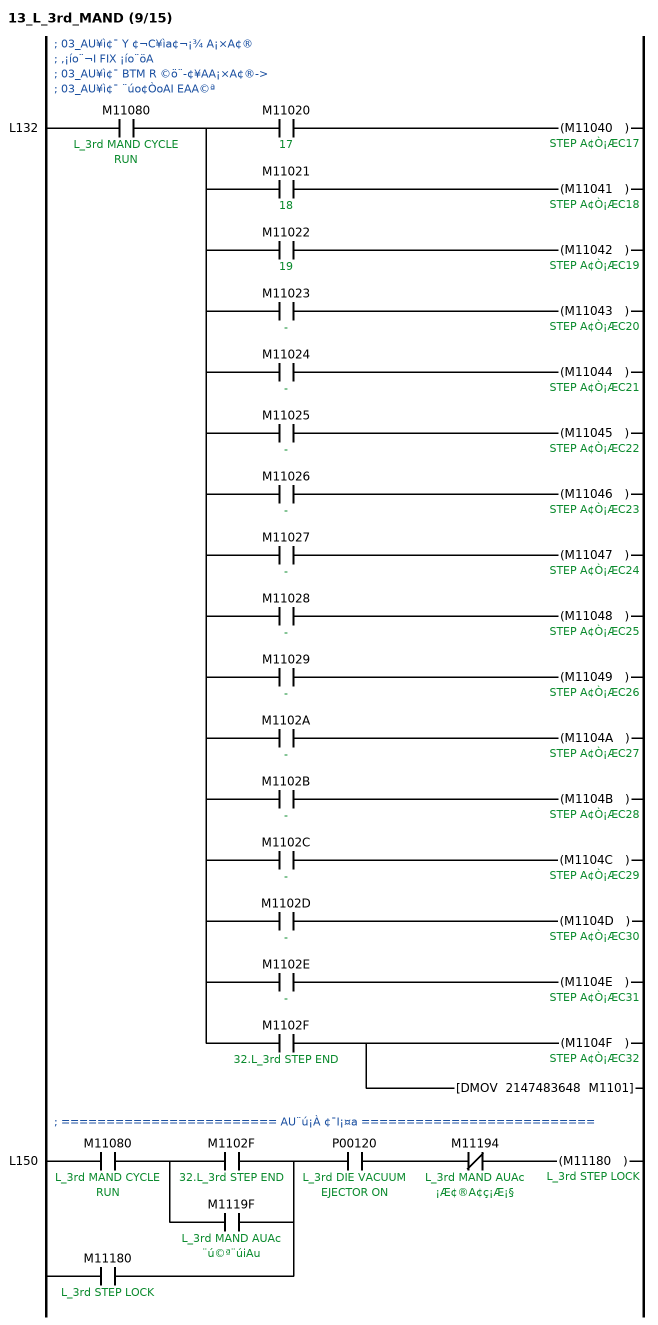
[picture p96: 13_L_3rd_MAND rungs L132-L150]
; L132
LOAD      M11080	// L_3rd MAND CYCLE RUN
MPUSH
AND       M11020	// 17
OUT       M11040	// STEP A¢Ò¡ÆC17
MLOAD
AND       M11021	// 18
OUT       M11041	// STEP A¢Ò¡ÆC18
MLOAD
AND       M11022	// 19
OUT       M11042	// STEP A¢Ò¡ÆC19
MLOAD
AND       M11023	// -
OUT       M11043	// STEP A¢Ò¡ÆC20
MLOAD
AND       M11024	// -
OUT       M11044	// STEP A¢Ò¡ÆC21
MLOAD
AND       M11025	// -
OUT       M11045	// STEP A¢Ò¡ÆC22
MLOAD
AND       M11026	// -
OUT       M11046	// STEP A¢Ò¡ÆC23
MLOAD
AND       M11027	// -
OUT       M11047	// STEP A¢Ò¡ÆC24
MLOAD
AND       M11028	// -
OUT       M11048	// STEP A¢Ò¡ÆC25
MLOAD
AND       M11029	// -
OUT       M11049	// STEP A¢Ò¡ÆC26
MLOAD
AND       M1102A	// -
OUT       M1104A	// STEP A¢Ò¡ÆC27
MLOAD
AND       M1102B	// -
OUT       M1104B	// STEP A¢Ò¡ÆC28
MLOAD
AND       M1102C	// -
OUT       M1104C	// STEP A¢Ò¡ÆC29
MLOAD
AND       M1102D	// -
OUT       M1104D	// STEP A¢Ò¡ÆC30
MLOAD
AND       M1102E	// -
OUT       M1104E	// STEP A¢Ò¡ÆC31
MPOP
AND       M1102F	// 32.L_3rd STEP END
OUT       M1104F	// STEP A¢Ò¡ÆC32
DMOV      2147483648 M1101
// output comment: 03_AU¥ì¢¯ Y ¢¬C¥ìa¢¬¡¾ A¡×A¢® ,¡ío¨¬I FIX ¡ío¨öA
// output comment: 03_AU¥ì¢¯ BTM R ©ö¨­¢¥AA¡×A¢®->
// output comment: 03_AU¥ì¢¯ ¨úo¢ÒoAI EAA©ª
// ======================== AU¨ú¡À ¢¯I¡¤a ==========================
; L150
LOAD      M11080	// L_3rd MAND CYCLE RUN
LOAD      M1102F	// 32.L_3rd STEP END
OR        M1119F	// L_3rd MAND AUAc ¨ú©ª¨úiAu
AND LOAD
OR        M11180	// L_3rd STEP LOCK
AND       P00120	// L_3rd DIE VACUUM EJECTOR ON
AND NOT   M11194	// L_3rd MAND AUAc ¡Æ¢®A¢ç¡Æ¡§
OUT       M11180	// L_3rd STEP LOCK

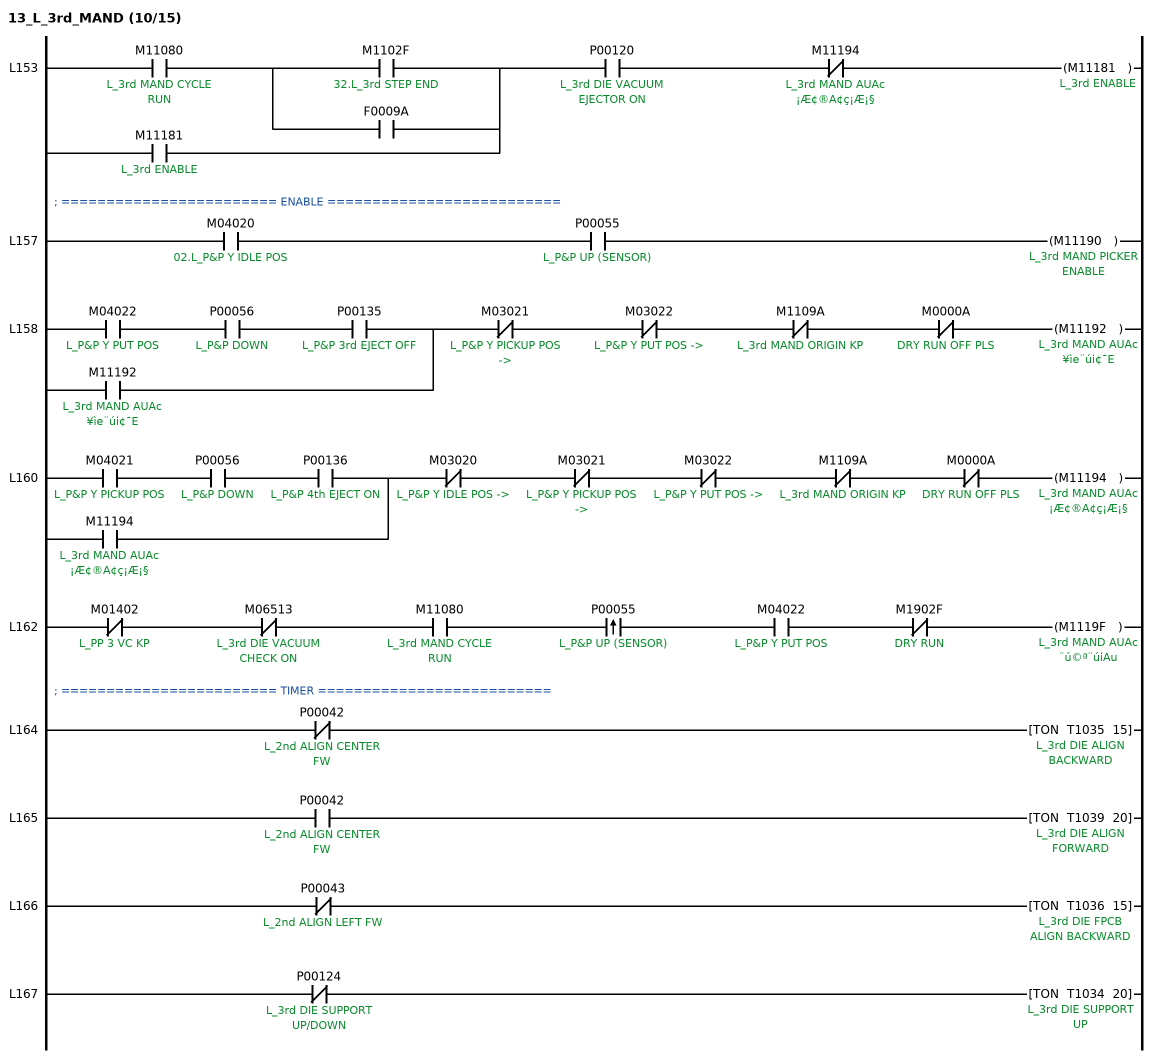
; L153
LOAD      M11080	// L_3rd MAND CYCLE RUN
LOAD      M1102F	// 32.L_3rd STEP END
OR        F0009A
AND LOAD
OR        M11181	// L_3rd ENABLE
AND       P00120	// L_3rd DIE VACUUM EJECTOR ON
AND NOT   M11194	// L_3rd MAND AUAc ¡Æ¢®A¢ç¡Æ¡§
OUT       M11181	// L_3rd ENABLE
// ======================== ENABLE ==========================
; L157
LOAD      M04020	// 02.L_P&P Y IDLE POS
AND       P00055	// L_P&P UP (SENSOR)
OUT       M11190	// L_3rd MAND PICKER ENABLE
; L158
LOAD      M04022	// L_P&P Y PUT POS
AND       P00056	// L_P&P DOWN
AND       P00135	// L_P&P 3rd EJECT OFF
OR        M11192	// L_3rd MAND AUAc ¥ìe¨úi¢¯E
AND NOT   M03021	// L_P&P Y PICKUP POS ->
AND NOT   M03022	// L_P&P Y PUT POS ->
AND NOT   M1109A	// L_3rd MAND ORIGIN KP
AND NOT   M0000A	// DRY RUN OFF PLS
OUT       M11192	// L_3rd MAND AUAc ¥ìe¨úi¢¯E
; L160
LOAD      M04021	// L_P&P Y PICKUP POS
AND       P00056	// L_P&P DOWN
AND       P00136	// L_P&P 4th EJECT ON
OR        M11194	// L_3rd MAND AUAc ¡Æ¢®A¢ç¡Æ¡§
AND NOT   M03020	// L_P&P Y IDLE POS ->
AND NOT   M03021	// L_P&P Y PICKUP POS ->
AND NOT   M03022	// L_P&P Y PUT POS ->
AND NOT   M1109A	// L_3rd MAND ORIGIN KP
AND NOT   M0000A	// DRY RUN OFF PLS
OUT       M11194	// L_3rd MAND AUAc ¡Æ¢®A¢ç¡Æ¡§
; L162
LOAD NOT  M01402	// L_PP 3 VC KP
AND NOT   M06513	// L_3rd DIE VACUUM CHECK ON
AND       M11080	// L_3rd MAND CYCLE RUN
ANDP      P00055	// L_P&P UP (SENSOR)
AND       M04022	// L_P&P Y PUT POS
AND NOT   M1902F	// DRY RUN
OUT       M1119F	// L_3rd MAND AUAc ¨ú©ª¨úiAu
// ======================== TIMER ==========================
; L164
LOAD NOT  P00042	// L_2nd ALIGN CENTER FW
TON       T1035 15	// L_3rd DIE ALIGN BACKWARD
; L165
LOAD      P00042	// L_2nd ALIGN CENTER FW
TON       T1039 20	// L_3rd DIE ALIGN FORWARD
; L166
LOAD NOT  P00043	// L_2nd ALIGN LEFT FW
TON       T1036 15	// L_3rd DIE FPCB ALIGN BACKWARD
; L167
LOAD NOT  P00124	// L_3rd DIE SUPPORT UP/DOWN
TON       T1034 20	// L_3rd DIE SUPPORT UP

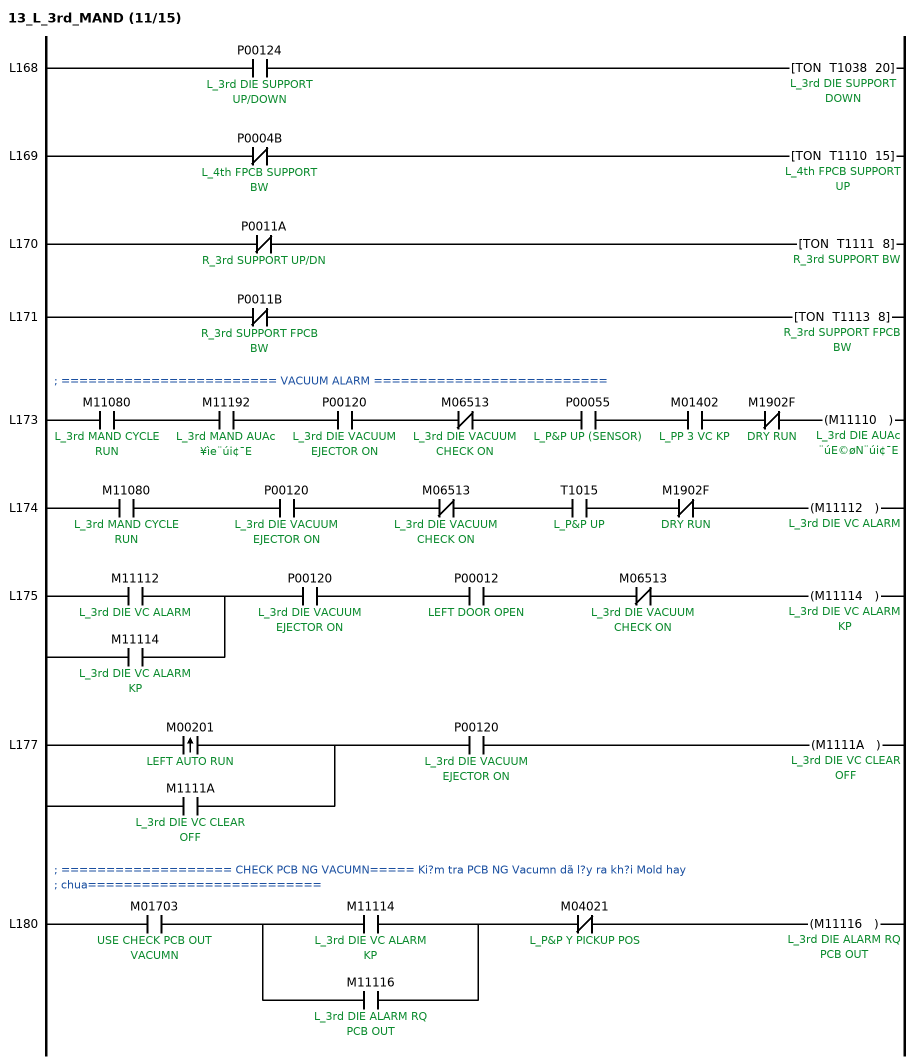
; L168
LOAD      P00124	// L_3rd DIE SUPPORT UP/DOWN
TON       T1038 20	// L_3rd DIE SUPPORT DOWN
; L169
LOAD NOT  P0004B	// L_4th FPCB SUPPORT BW
TON       T1110 15	// L_4th FPCB SUPPORT UP
; L170
LOAD NOT  P0011A	// R_3rd SUPPORT UP/DN
TON       T1111 8	// R_3rd SUPPORT BW
; L171
LOAD NOT  P0011B	// R_3rd SUPPORT FPCB BW
TON       T1113 8	// R_3rd SUPPORT FPCB BW
// ======================== VACUUM ALARM ==========================
; L173
LOAD      M11080	// L_3rd MAND CYCLE RUN
AND       M11192	// L_3rd MAND AUAc ¥ìe¨úi¢¯E
AND       P00120	// L_3rd DIE VACUUM EJECTOR ON
AND NOT   M06513	// L_3rd DIE VACUUM CHECK ON
AND       P00055	// L_P&P UP (SENSOR)
AND       M01402	// L_PP 3 VC KP
AND NOT   M1902F	// DRY RUN
OUT       M11110	// L_3rd DIE AUAc ¨úE©øN¨úi¢¯E
; L174
LOAD      M11080	// L_3rd MAND CYCLE RUN
AND       P00120	// L_3rd DIE VACUUM EJECTOR ON
AND NOT   M06513	// L_3rd DIE VACUUM CHECK ON
AND       T1015	// L_P&P UP
AND NOT   M1902F	// DRY RUN
OUT       M11112	// L_3rd DIE VC ALARM
; L175
LOAD      M11112	// L_3rd DIE VC ALARM
OR        M11114	// L_3rd DIE VC ALARM KP
AND       P00120	// L_3rd DIE VACUUM EJECTOR ON
AND       P00012	// LEFT DOOR OPEN
AND NOT   M06513	// L_3rd DIE VACUUM CHECK ON
OUT       M11114	// L_3rd DIE VC ALARM KP
; L177
LOADP     M00201	// LEFT AUTO RUN
OR        M1111A	// L_3rd DIE VC CLEAR OFF
AND       P00120	// L_3rd DIE VACUUM EJECTOR ON
OUT       M1111A	// L_3rd DIE VC CLEAR OFF
// =================== CHECK PCB NG VACUMN===== Ki?m tra PCB NG Vacumn dã l?y ra kh?i Mold hay chua==========================
; L180
LOAD      M01703	// USE CHECK PCB OUT VACUMN
LOAD      M11114	// L_3rd DIE VC ALARM KP
OR        M11116	// L_3rd DIE ALARM RQ PCB OUT
AND LOAD
AND NOT   M04021	// L_P&P Y PICKUP POS
OUT       M11116	// L_3rd DIE ALARM RQ PCB OUT

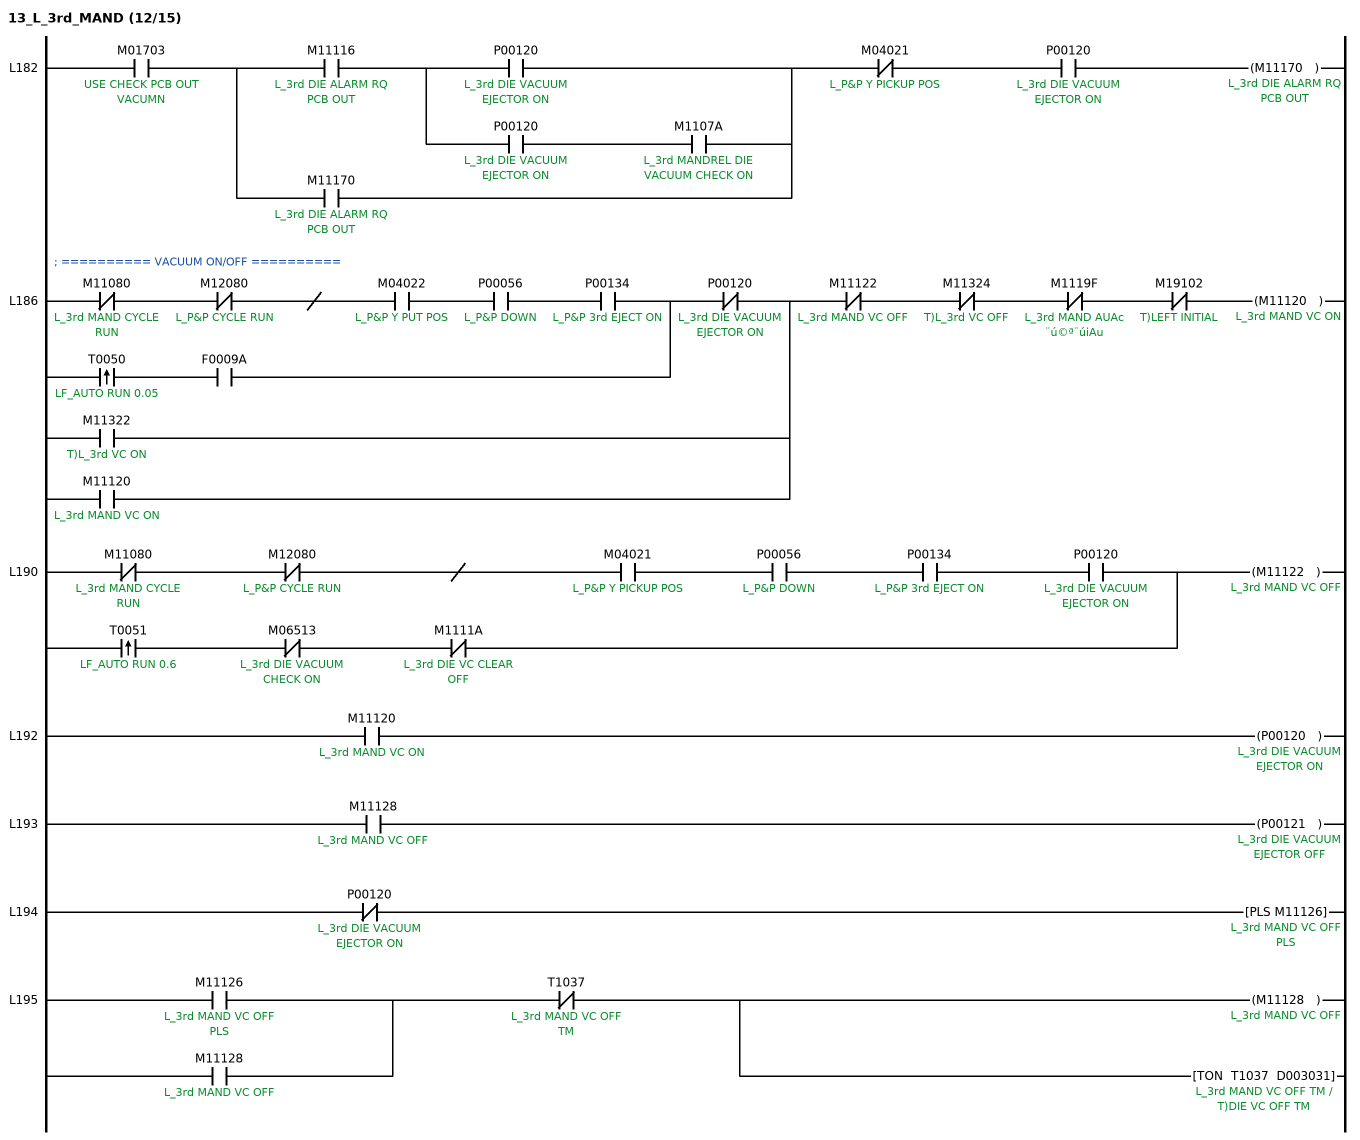
; L182
LOAD      M01703	// USE CHECK PCB OUT VACUMN
LOAD      M11116	// L_3rd DIE ALARM RQ PCB OUT
LOAD      P00120	// L_3rd DIE VACUUM EJECTOR ON
LOAD      P00120	// L_3rd DIE VACUUM EJECTOR ON
AND       M1107A	// L_3rd MANDREL DIE VACUUM CHECK ON
OR LOAD
AND LOAD
OR        M11170	// L_3rd DIE ALARM RQ PCB OUT
AND LOAD
AND NOT   M04021	// L_P&P Y PICKUP POS
AND       P00120	// L_3rd DIE VACUUM EJECTOR ON
OUT       M11170	// L_3rd DIE ALARM RQ PCB OUT
// ========== VACUUM ON/OFF ==========
; L186
LOAD NOT  M11080	// L_3rd MAND CYCLE RUN
AND NOT   M12080	// L_P&P CYCLE RUN
NOT
AND       M04022	// L_P&P Y PUT POS
AND       P00056	// L_P&P DOWN
AND       P00134	// L_P&P 3rd EJECT ON
LOADP     T0050	// LF_AUTO RUN 0.05
AND       F0009A
OR LOAD
AND NOT   P00120	// L_3rd DIE VACUUM EJECTOR ON
OR        M11322	// T)L_3rd VC ON
OR        M11120	// L_3rd MAND VC ON
AND NOT   M11122	// L_3rd MAND VC OFF
AND NOT   M11324	// T)L_3rd VC OFF
AND NOT   M1119F	// L_3rd MAND AUAc ¨ú©ª¨úiAu
AND NOT   M19102	// T)LEFT INITIAL
OUT       M11120	// L_3rd MAND VC ON
; L190
LOAD NOT  M11080	// L_3rd MAND CYCLE RUN
AND NOT   M12080	// L_P&P CYCLE RUN
NOT
AND       M04021	// L_P&P Y PICKUP POS
AND       P00056	// L_P&P DOWN
AND       P00134	// L_P&P 3rd EJECT ON
AND       P00120	// L_3rd DIE VACUUM EJECTOR ON
LOADP     T0051	// LF_AUTO RUN 0.6
AND NOT   M06513	// L_3rd DIE VACUUM CHECK ON
AND NOT   M1111A	// L_3rd DIE VC CLEAR OFF
OR LOAD
OUT       M11122	// L_3rd MAND VC OFF
; L192
LOAD      M11120	// L_3rd MAND VC ON
OUT       P00120	// L_3rd DIE VACUUM EJECTOR ON
; L193
LOAD      M11128	// L_3rd MAND VC OFF
OUT       P00121	// L_3rd DIE VACUUM EJECTOR OFF
; L194
LOAD NOT  P00120	// L_3rd DIE VACUUM EJECTOR ON
OUTP      M11126	// L_3rd MAND VC OFF PLS
; L195
LOAD      M11126	// L_3rd MAND VC OFF PLS
OR        M11128	// L_3rd MAND VC OFF
AND NOT   T1037	// L_3rd MAND VC OFF TM
OUT       M11128	// L_3rd MAND VC OFF
TON       T1037 D003031	// L_3rd MAND VC OFF TM / T)DIE VC OFF TM

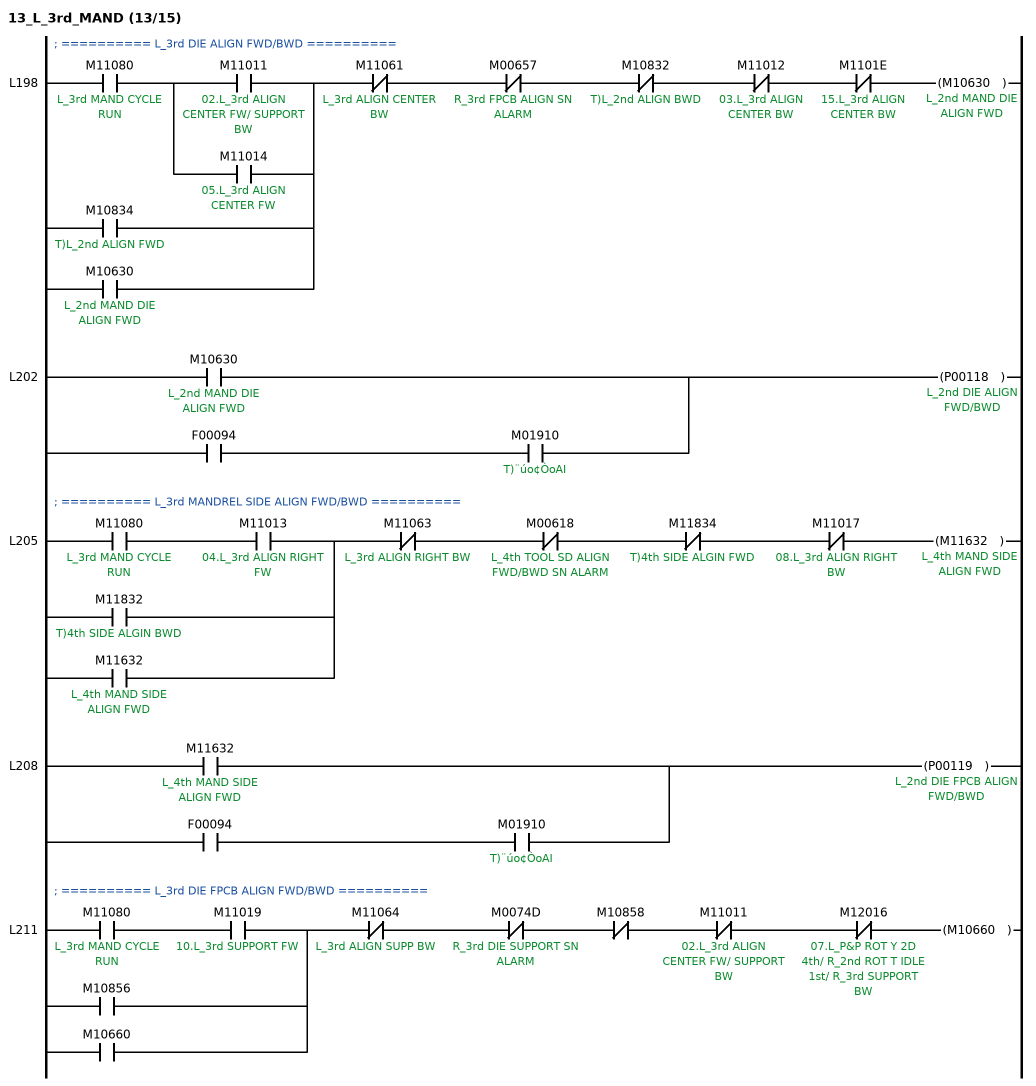
// ========== L_3rd DIE ALIGN FWD/BWD ==========
; L198
LOAD      M11080	// L_3rd MAND CYCLE RUN
LOAD      M11011	// 02.L_3rd ALIGN CENTER FW/ SUPPORT BW
OR        M11014	// 05.L_3rd ALIGN CENTER FW
AND LOAD
OR        M10834	// T)L_2nd ALIGN FWD
OR        M10630	// L_2nd MAND DIE ALIGN FWD
AND NOT   M11061	// L_3rd ALIGN CENTER BW
AND NOT   M00657	// R_3rd FPCB ALIGN SN ALARM
AND NOT   M10832	// T)L_2nd ALIGN BWD
AND NOT   M11012	// 03.L_3rd ALIGN CENTER BW
AND NOT   M1101E	// 15.L_3rd ALIGN CENTER BW
OUT       M10630	// L_2nd MAND DIE ALIGN FWD
; L202
LOAD      M10630	// L_2nd MAND DIE ALIGN FWD
LOAD      F00094
AND       M01910	// T)¨úo¢ÒoAI
OR LOAD
OUT       P00118	// L_2nd DIE ALIGN FWD/BWD
// ========== L_3rd MANDREL SIDE ALIGN FWD/BWD ==========
; L205
LOAD      M11080	// L_3rd MAND CYCLE RUN
AND       M11013	// 04.L_3rd ALIGN RIGHT FW
OR        M11832	// T)4th SIDE ALGIN BWD
OR        M11632	// L_4th MAND SIDE ALIGN FWD
AND NOT   M11063	// L_3rd ALIGN RIGHT BW
AND NOT   M00618	// L_4th TOOL SD ALIGN FWD/BWD SN ALARM
AND NOT   M11834	// T)4th SIDE ALGIN FWD
AND NOT   M11017	// 08.L_3rd ALIGN RIGHT BW
OUT       M11632	// L_4th MAND SIDE ALIGN FWD
; L208
LOAD      M11632	// L_4th MAND SIDE ALIGN FWD
LOAD      F00094
AND       M01910	// T)¨úo¢ÒoAI
OR LOAD
OUT       P00119	// L_2nd DIE FPCB ALIGN FWD/BWD
// ========== L_3rd DIE FPCB ALIGN FWD/BWD ==========
; L211
LOAD      M11080	// L_3rd MAND CYCLE RUN
AND       M11019	// 10.L_3rd SUPPORT FW
OR        M10856
OR        M10660
AND NOT   M11064	// L_3rd ALIGN SUPP BW
AND NOT   M0074D	// R_3rd DIE SUPPORT SN ALARM
AND NOT   M10858
AND NOT   M11011	// 02.L_3rd ALIGN CENTER FW/ SUPPORT BW
AND NOT   M12016	// 07.L_P&P ROT Y 2D 4th/ R_2nd ROT T IDLE 1st/ R_3rd SUPPORT BW
OUT       M10660

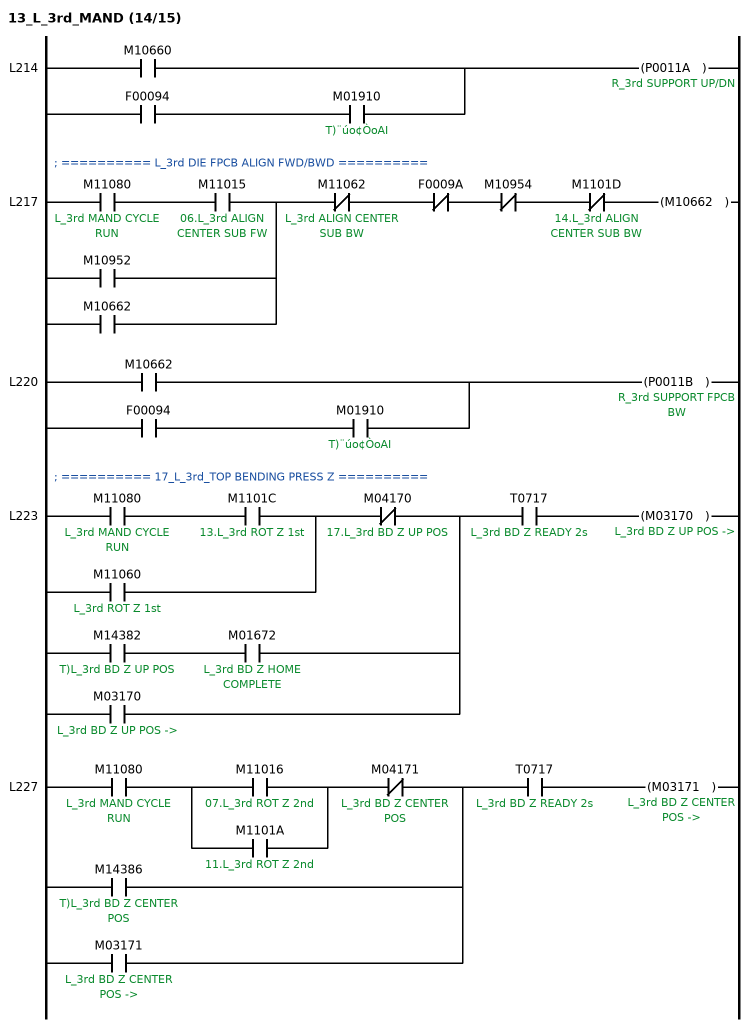
; L214
LOAD      M10660
LOAD      F00094
AND       M01910	// T)¨úo¢ÒoAI
OR LOAD
OUT       P0011A	// R_3rd SUPPORT UP/DN
// ========== L_3rd DIE FPCB ALIGN FWD/BWD ==========
; L217
LOAD      M11080	// L_3rd MAND CYCLE RUN
AND       M11015	// 06.L_3rd ALIGN CENTER SUB FW
OR        M10952
OR        M10662
AND NOT   M11062	// L_3rd ALIGN CENTER SUB BW
AND NOT   F0009A
AND NOT   M10954
AND NOT   M1101D	// 14.L_3rd ALIGN CENTER SUB BW
OUT       M10662
; L220
LOAD      M10662
LOAD      F00094
AND       M01910	// T)¨úo¢ÒoAI
OR LOAD
OUT       P0011B	// R_3rd SUPPORT FPCB BW
// ========== 17_L_3rd_TOP BENDING PRESS Z ==========
; L223
LOAD      M11080	// L_3rd MAND CYCLE RUN
AND       M1101C	// 13.L_3rd ROT Z 1st
OR        M11060	// L_3rd ROT Z 1st
AND NOT   M04170	// 17.L_3rd BD Z UP POS
LOAD      M14382	// T)L_3rd BD Z UP POS
AND       M01672	// L_3rd BD Z HOME COMPLETE
OR LOAD
OR        M03170	// L_3rd BD Z UP POS ->
AND       T0717	// L_3rd BD Z READY 2s
OUT       M03170	// L_3rd BD Z UP POS ->
; L227
LOAD      M11080	// L_3rd MAND CYCLE RUN
LOAD      M11016	// 07.L_3rd ROT Z 2nd
OR        M1101A	// 11.L_3rd ROT Z 2nd
AND LOAD
AND NOT   M04171	// L_3rd BD Z CENTER POS
OR        M14386	// T)L_3rd BD Z CENTER POS
OR        M03171	// L_3rd BD Z CENTER POS ->
AND       T0717	// L_3rd BD Z READY 2s
OUT       M03171	// L_3rd BD Z CENTER POS ->

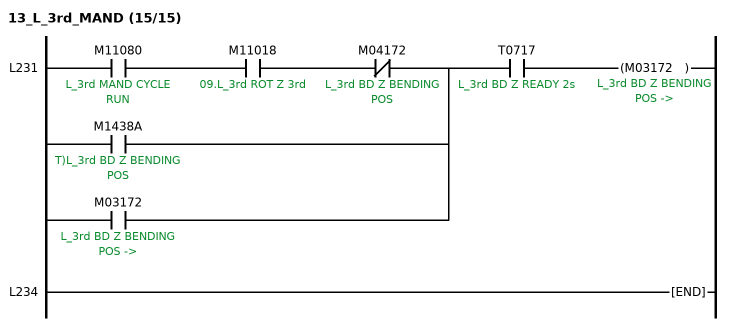
; L231
LOAD      M11080	// L_3rd MAND CYCLE RUN
AND       M11018	// 09.L_3rd ROT Z 3rd
AND NOT   M04172	// L_3rd BD Z BENDING POS
OR        M1438A	// T)L_3rd BD Z BENDING POS
OR        M03172	// L_3rd BD Z BENDING POS ->
AND       T0717	// L_3rd BD Z READY 2s
OUT       M03172	// L_3rd BD Z BENDING POS ->
; L234
END

PROGRAM 14_L_TOOL (task: ¨ö¨¬A¥ì CA¡¤I¡¾¡¿¡¤¡Í)

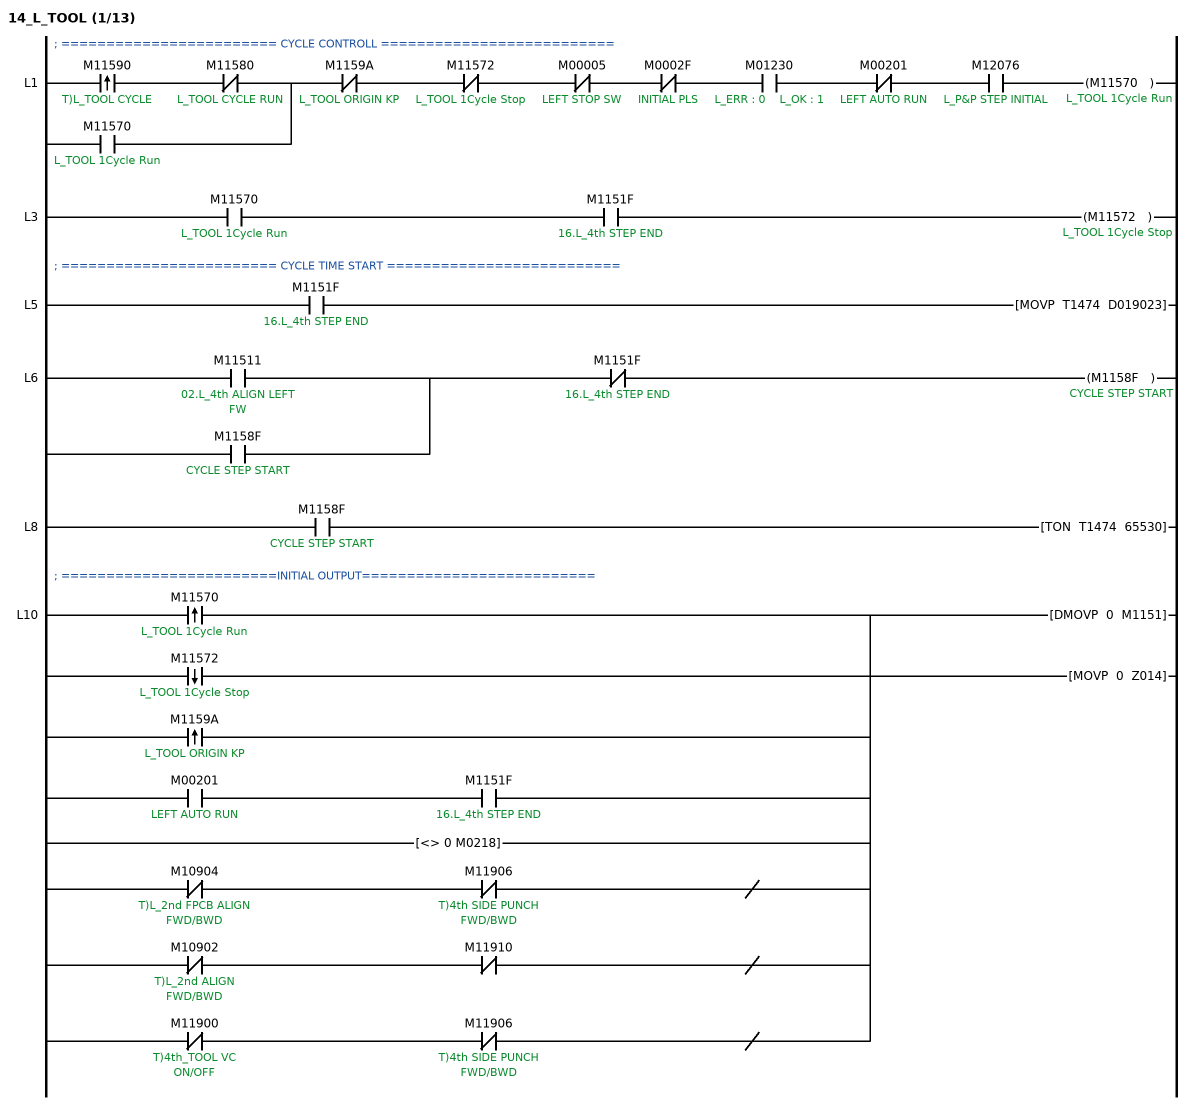
// ======================== CYCLE CONTROLL ==========================
; L1
LOADP     M11590	// T)L_TOOL CYCLE
AND NOT   M11580	// L_TOOL CYCLE RUN
OR        M11570	// L_TOOL 1Cycle Run
AND NOT   M1159A	// L_TOOL ORIGIN KP
AND NOT   M11572	// L_TOOL 1Cycle Stop
AND NOT   M00005	// LEFT STOP SW
AND NOT   M0002F	// INITIAL PLS
AND       M01230	// L_ERR : 0    L_OK : 1
AND NOT   M00201	// LEFT AUTO RUN
AND       M12076	// L_P&P STEP INITIAL
OUT       M11570	// L_TOOL 1Cycle Run
; L3
LOAD      M11570	// L_TOOL 1Cycle Run
AND       M1151F	// 16.L_4th STEP END
OUT       M11572	// L_TOOL 1Cycle Stop
// ======================== CYCLE TIME START ==========================
; L5
LOAD      M1151F	// 16.L_4th STEP END
MOVP      T1474 D019023
; L6
LOAD      M11511	// 02.L_4th ALIGN LEFT FW
OR        M1158F	// CYCLE STEP START
AND NOT   M1151F	// 16.L_4th STEP END
OUT       M1158F	// CYCLE STEP START
; L8
LOAD      M1158F	// CYCLE STEP START
TON       T1474 65530
// ========================INITIAL OUTPUT==========================
; L10
LOADP     M11570	// L_TOOL 1Cycle Run
ORN       M11572	// L_TOOL 1Cycle Stop
ORP       M1159A	// L_TOOL ORIGIN KP
LOAD      M00201	// LEFT AUTO RUN
AND       M1151F	// 16.L_4th STEP END
OR LOAD
OR<>      0 M0218
LOAD NOT  M10904	// T)L_2nd FPCB ALIGN FWD/BWD
AND NOT   M11906	// T)4th SIDE PUNCH FWD/BWD
NOT
OR LOAD
LOAD NOT  M10902	// T)L_2nd ALIGN FWD/BWD
AND NOT   M11910
NOT
OR LOAD
LOAD NOT  M11900	// T)4th_TOOL VC ON/OFF
AND NOT   M11906	// T)4th SIDE PUNCH FWD/BWD
NOT
OR LOAD
DMOVP     0 M1151
MOVP      0 Z014

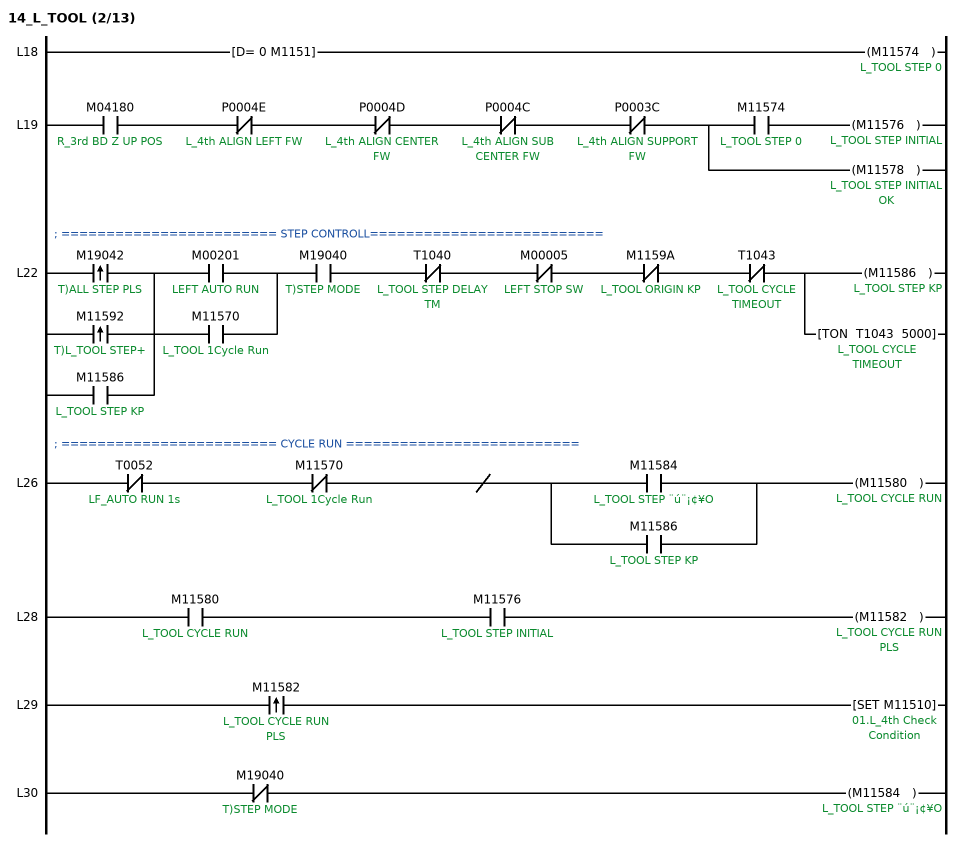
; L18
LOADD=    0 M1151
OUT       M11574	// L_TOOL STEP 0
; L19
LOAD      M04180	// R_3rd BD Z UP POS
AND NOT   P0004E	// L_4th ALIGN LEFT FW
AND NOT   P0004D	// L_4th ALIGN CENTER FW
AND NOT   P0004C	// L_4th ALIGN SUB CENTER FW
AND NOT   P0003C	// L_4th ALIGN SUPPORT FW
MPUSH
AND       M11574	// L_TOOL STEP 0
OUT       M11576	// L_TOOL STEP INITIAL
MPOP
OUT       M11578	// L_TOOL STEP INITIAL OK
// ======================== STEP CONTROLL==========================
; L22
LOADP     M19042	// T)ALL STEP PLS
ORP       M11592	// T)L_TOOL STEP+
OR        M11586	// L_TOOL STEP KP
LOAD      M00201	// LEFT AUTO RUN
OR        M11570	// L_TOOL 1Cycle Run
AND LOAD
AND       M19040	// T)STEP MODE
AND NOT   T1040	// L_TOOL STEP DELAY TM
AND NOT   M00005	// LEFT STOP SW
AND NOT   M1159A	// L_TOOL ORIGIN KP
AND NOT   T1043	// L_TOOL CYCLE TIMEOUT
OUT       M11586	// L_TOOL STEP KP
TON       T1043 5000	// L_TOOL CYCLE TIMEOUT
// ======================== CYCLE RUN ==========================
; L26
LOAD NOT  T0052	// LF_AUTO RUN 1s
AND NOT   M11570	// L_TOOL 1Cycle Run
NOT
LOAD      M11584	// L_TOOL STEP ¨ú¨¡¢¥O
OR        M11586	// L_TOOL STEP KP
AND LOAD
OUT       M11580	// L_TOOL CYCLE RUN
; L28
LOAD      M11580	// L_TOOL CYCLE RUN
AND       M11576	// L_TOOL STEP INITIAL
OUT       M11582	// L_TOOL CYCLE RUN PLS
; L29
LOADP     M11582	// L_TOOL CYCLE RUN PLS
SET       M11510	// 01.L_4th Check Condition
; L30
LOAD NOT  M19040	// T)STEP MODE
OUT       M11584	// L_TOOL STEP ¨ú¨¡¢¥O

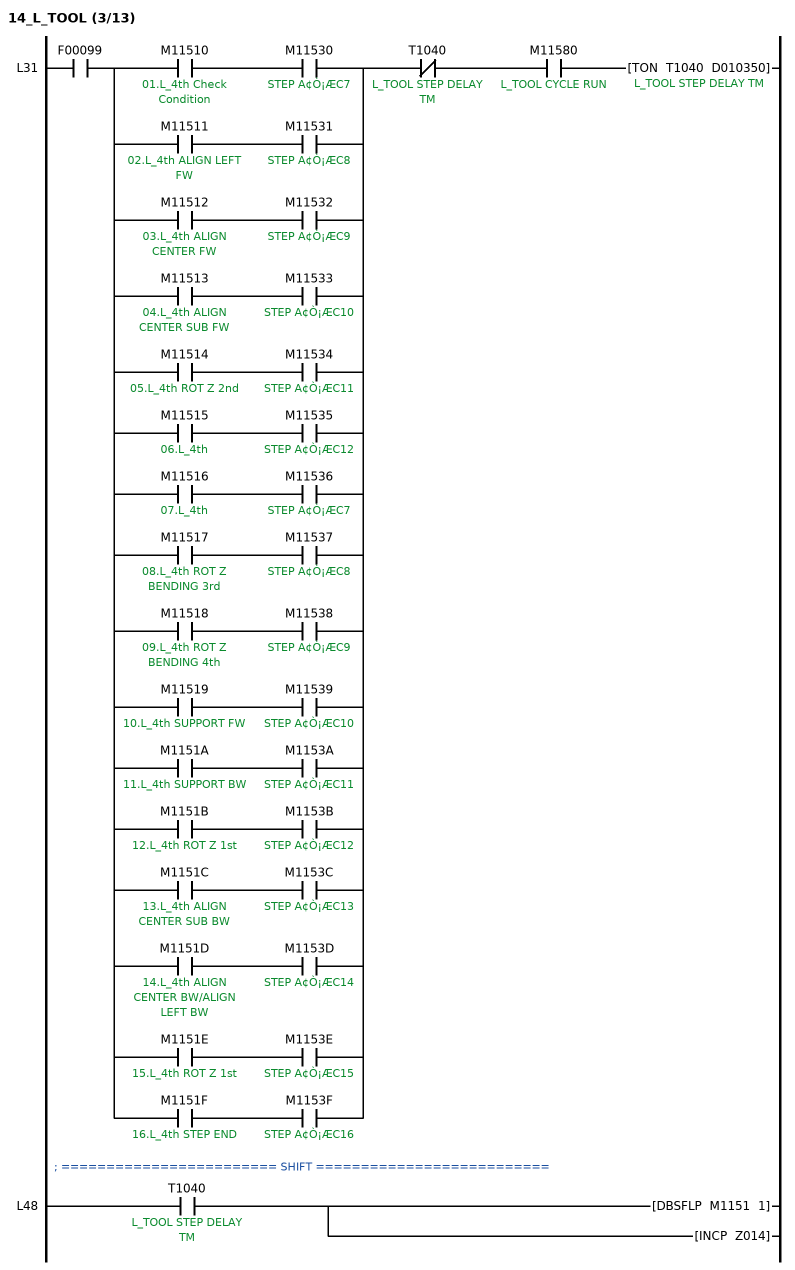
; L31
LOAD      F00099
LOAD      M11510	// 01.L_4th Check Condition
AND       M11530	// STEP A¢Ò¡ÆC7
LOAD      M11511	// 02.L_4th ALIGN LEFT FW
AND       M11531	// STEP A¢Ò¡ÆC8
OR LOAD
LOAD      M11512	// 03.L_4th ALIGN CENTER FW
AND       M11532	// STEP A¢Ò¡ÆC9
OR LOAD
LOAD      M11513	// 04.L_4th ALIGN CENTER SUB FW
AND       M11533	// STEP A¢Ò¡ÆC10
OR LOAD
LOAD      M11514	// 05.L_4th ROT Z 2nd
AND       M11534	// STEP A¢Ò¡ÆC11
OR LOAD
LOAD      M11515	// 06.L_4th 
AND       M11535	// STEP A¢Ò¡ÆC12
OR LOAD
LOAD      M11516	// 07.L_4th 
AND       M11536	// STEP A¢Ò¡ÆC7
OR LOAD
LOAD      M11517	// 08.L_4th ROT Z BENDING 3rd
AND       M11537	// STEP A¢Ò¡ÆC8
OR LOAD
LOAD      M11518	// 09.L_4th ROT Z BENDING 4th
AND       M11538	// STEP A¢Ò¡ÆC9
OR LOAD
LOAD      M11519	// 10.L_4th SUPPORT FW
AND       M11539	// STEP A¢Ò¡ÆC10
OR LOAD
LOAD      M1151A	// 11.L_4th SUPPORT BW
AND       M1153A	// STEP A¢Ò¡ÆC11
OR LOAD
LOAD      M1151B	// 12.L_4th ROT Z 1st
AND       M1153B	// STEP A¢Ò¡ÆC12
OR LOAD
LOAD      M1151C	// 13.L_4th ALIGN CENTER SUB BW
AND       M1153C	// STEP A¢Ò¡ÆC13
OR LOAD
LOAD      M1151D	// 14.L_4th ALIGN CENTER BW/ALIGN LEFT BW
AND       M1153D	// STEP A¢Ò¡ÆC14
OR LOAD
LOAD      M1151E	// 15.L_4th ROT Z 1st
AND       M1153E	// STEP A¢Ò¡ÆC15
OR LOAD
LOAD      M1151F	// 16.L_4th STEP END
AND       M1153F	// STEP A¢Ò¡ÆC16
OR LOAD
AND LOAD
AND NOT   T1040	// L_TOOL STEP DELAY TM
AND       M11580	// L_TOOL CYCLE RUN
TON       T1040 D010350	// L_TOOL STEP DELAY TM
// ======================== SHIFT ==========================
; L48
LOAD      T1040	// L_TOOL STEP DELAY TM
DBSFLP    M1151 1
INCP      Z014

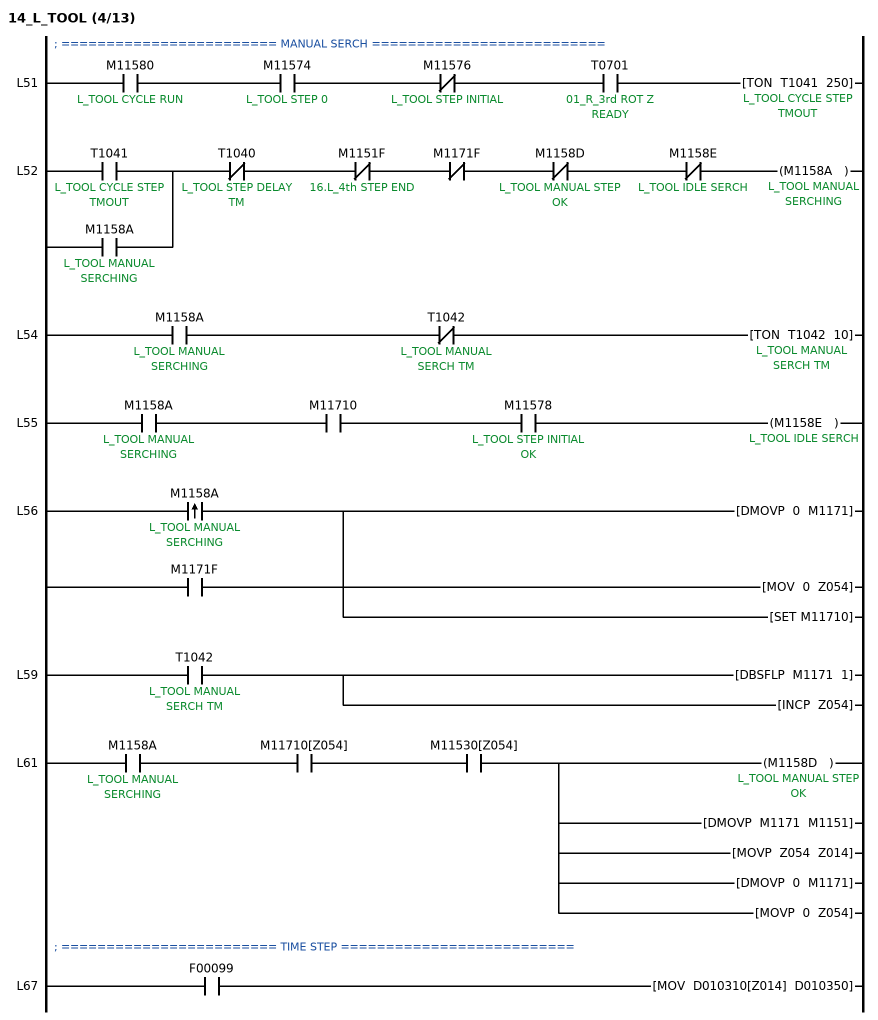
// ======================== MANUAL SERCH ==========================
; L51
LOAD      M11580	// L_TOOL CYCLE RUN
AND       M11574	// L_TOOL STEP 0
AND NOT   M11576	// L_TOOL STEP INITIAL
AND       T0701	// 01_R_3rd ROT Z READY
TON       T1041 250	// L_TOOL CYCLE STEP TMOUT
; L52
LOAD      T1041	// L_TOOL CYCLE STEP TMOUT
OR        M1158A	// L_TOOL MANUAL SERCHING
AND NOT   T1040	// L_TOOL STEP DELAY TM
AND NOT   M1151F	// 16.L_4th STEP END
AND NOT   M1171F
AND NOT   M1158D	// L_TOOL MANUAL STEP OK
AND NOT   M1158E	// L_TOOL IDLE SERCH
OUT       M1158A	// L_TOOL MANUAL SERCHING
; L54
LOAD      M1158A	// L_TOOL MANUAL SERCHING
AND NOT   T1042	// L_TOOL MANUAL SERCH TM
TON       T1042 10	// L_TOOL MANUAL SERCH TM
; L55
LOAD      M1158A	// L_TOOL MANUAL SERCHING
AND       M11710
AND       M11578	// L_TOOL STEP INITIAL OK
OUT       M1158E	// L_TOOL IDLE SERCH
; L56
LOADP     M1158A	// L_TOOL MANUAL SERCHING
OR        M1171F
DMOVP     0 M1171
MOV       0 Z054
SET       M11710
; L59
LOAD      T1042	// L_TOOL MANUAL SERCH TM
DBSFLP    M1171 1
INCP      Z054
; L61
LOAD      M1158A	// L_TOOL MANUAL SERCHING
AND       M11710[Z054]
AND       M11530[Z054]
OUT       M1158D	// L_TOOL MANUAL STEP OK
DMOVP     M1171 M1151
MOVP      Z054 Z014
DMOVP     0 M1171
MOVP      0 Z054
// ======================== TIME STEP ==========================
; L67
LOAD      F00099
MOV       D010310[Z014] D010350

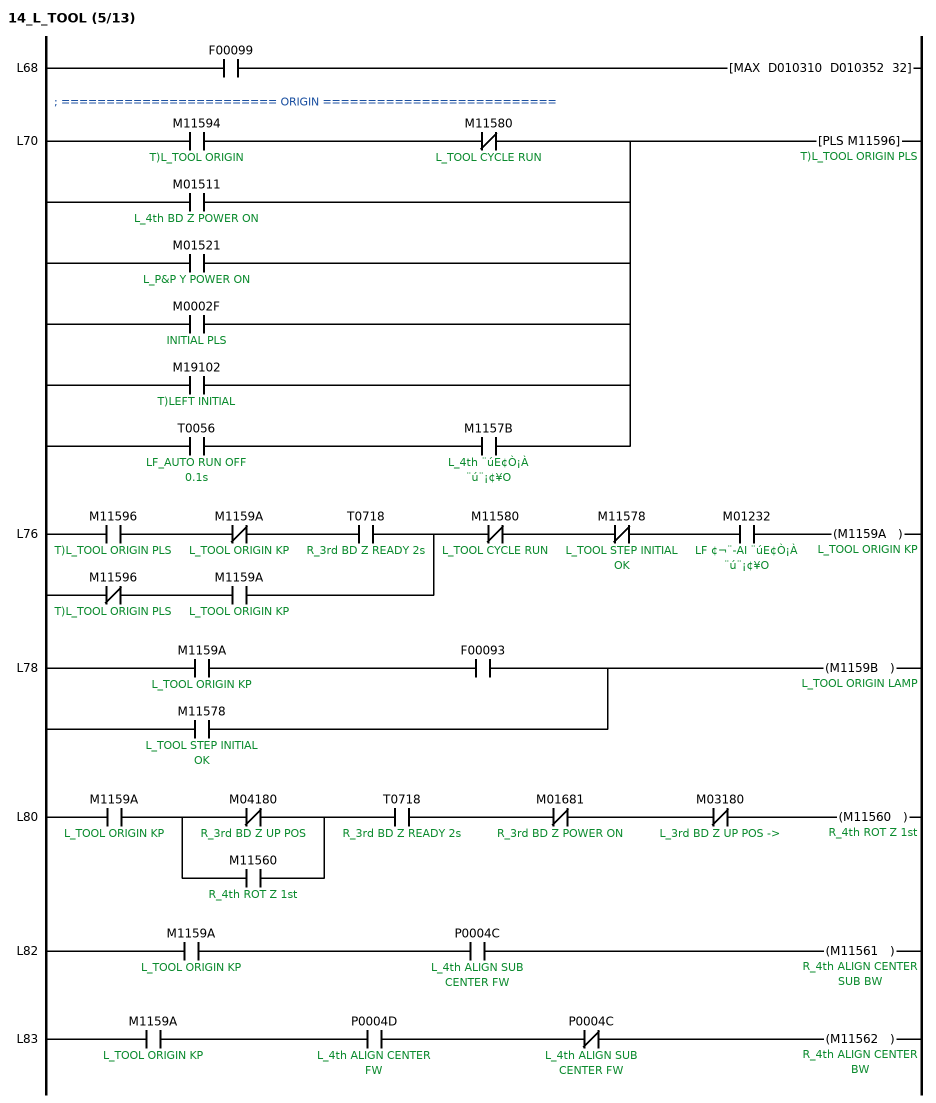
; L68
LOAD      F00099
MAX       D010310 D010352 32
// ======================== ORIGIN ==========================
; L70
LOAD      M11594	// T)L_TOOL ORIGIN
AND NOT   M11580	// L_TOOL CYCLE RUN
OR        M01511	// L_4th BD Z POWER ON
OR        M01521	// L_P&P Y POWER ON
OR        M0002F	// INITIAL PLS
OR        M19102	// T)LEFT INITIAL
LOAD      T0056	// LF_AUTO RUN OFF 0.1s
AND       M1157B	// L_4th ¨úE¢Ò¡À ¨ú¨¡¢¥O
OR LOAD
OUTP      M11596	// T)L_TOOL ORIGIN PLS
; L76
LOAD      M11596	// T)L_TOOL ORIGIN PLS
AND NOT   M1159A	// L_TOOL ORIGIN KP
AND       T0718	// R_3rd BD Z READY 2s
LOAD NOT  M11596	// T)L_TOOL ORIGIN PLS
AND       M1159A	// L_TOOL ORIGIN KP
OR LOAD
AND NOT   M11580	// L_TOOL CYCLE RUN
AND NOT   M11578	// L_TOOL STEP INITIAL OK
AND       M01232	// LF ¢¬¨­AI ¨úE¢Ò¡À ¨ú¨¡¢¥O
OUT       M1159A	// L_TOOL ORIGIN KP
; L78
LOAD      M1159A	// L_TOOL ORIGIN KP
AND       F00093
OR        M11578	// L_TOOL STEP INITIAL OK
OUT       M1159B	// L_TOOL ORIGIN LAMP
; L80
LOAD      M1159A	// L_TOOL ORIGIN KP
LOAD NOT  M04180	// R_3rd BD Z UP POS
OR        M11560	// R_4th ROT Z 1st
AND LOAD
AND       T0718	// R_3rd BD Z READY 2s
AND NOT   M01681	// R_3rd BD Z POWER ON
AND NOT   M03180	// L_3rd BD Z UP POS ->
OUT       M11560	// R_4th ROT Z 1st
; L82
LOAD      M1159A	// L_TOOL ORIGIN KP
AND       P0004C	// L_4th ALIGN SUB CENTER FW
OUT       M11561	// R_4th ALIGN CENTER SUB BW
; L83
LOAD      M1159A	// L_TOOL ORIGIN KP
AND       P0004D	// L_4th ALIGN CENTER FW
AND NOT   P0004C	// L_4th ALIGN SUB CENTER FW
OUT       M11562	// R_4th ALIGN CENTER BW

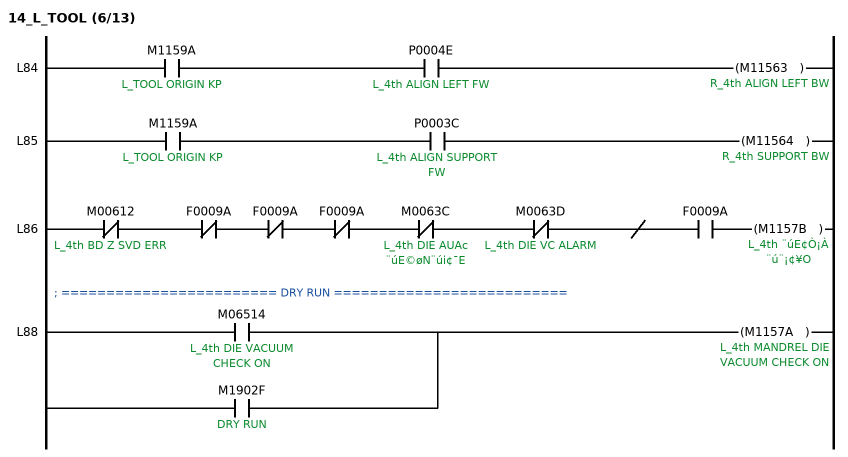
; L84
LOAD      M1159A	// L_TOOL ORIGIN KP
AND       P0004E	// L_4th ALIGN LEFT FW
OUT       M11563	// R_4th ALIGN LEFT BW
; L85
LOAD      M1159A	// L_TOOL ORIGIN KP
AND       P0003C	// L_4th ALIGN SUPPORT FW
OUT       M11564	// R_4th SUPPORT BW
; L86
LOAD NOT  M00612	// L_4th BD Z SVD ERR
AND NOT   F0009A
AND NOT   F0009A
AND NOT   F0009A
AND NOT   M0063C	// L_4th DIE AUAc ¨úE©øN¨úi¢¯E
AND NOT   M0063D	// L_4th DIE VC ALARM
NOT
AND       F0009A
OUT       M1157B	// L_4th ¨úE¢Ò¡À ¨ú¨¡¢¥O
// ======================== DRY RUN ==========================
; L88
LOAD      M06514	// L_4th DIE VACUUM CHECK ON
OR        M1902F	// DRY RUN
OUT       M1157A	// L_4th MANDREL DIE VACUUM CHECK ON

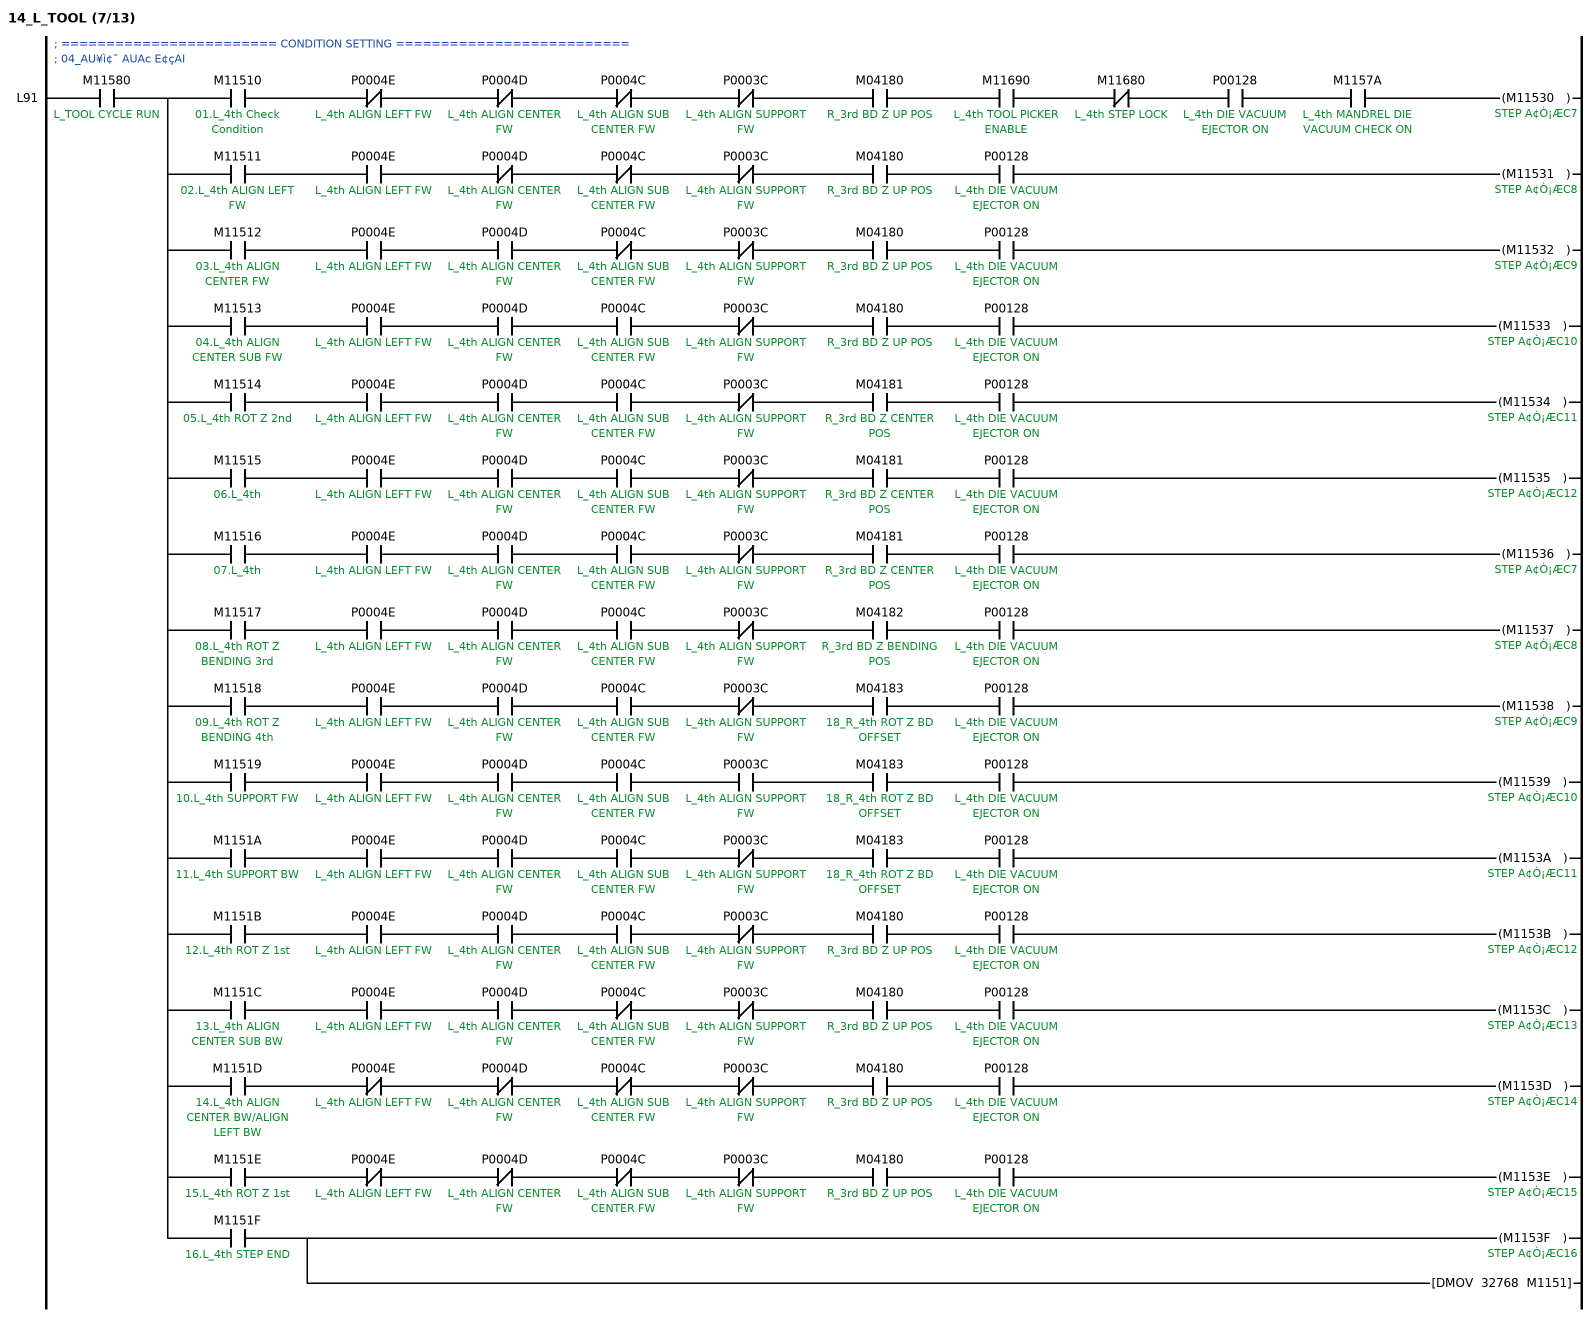
// ======================== CONDITION SETTING ==========================
; L91
LOAD      M11580	// L_TOOL CYCLE RUN
MPUSH
AND       M11510	// 01.L_4th Check Condition
AND NOT   P0004E	// L_4th ALIGN LEFT FW
AND NOT   P0004D	// L_4th ALIGN CENTER FW
AND NOT   P0004C	// L_4th ALIGN SUB CENTER FW
AND NOT   P0003C	// L_4th ALIGN SUPPORT FW
AND       M04180	// R_3rd BD Z UP POS
AND       M11690	// L_4th TOOL PICKER ENABLE
AND NOT   M11680	// L_4th STEP LOCK
AND       P00128	// L_4th DIE VACUUM EJECTOR ON
AND       M1157A	// L_4th MANDREL DIE VACUUM CHECK ON
OUT       M11530	// STEP A¢Ò¡ÆC7
MLOAD
AND       M11511	// 02.L_4th ALIGN LEFT FW
AND       P0004E	// L_4th ALIGN LEFT FW
AND NOT   P0004D	// L_4th ALIGN CENTER FW
AND NOT   P0004C	// L_4th ALIGN SUB CENTER FW
AND NOT   P0003C	// L_4th ALIGN SUPPORT FW
AND       M04180	// R_3rd BD Z UP POS
AND       P00128	// L_4th DIE VACUUM EJECTOR ON
OUT       M11531	// STEP A¢Ò¡ÆC8
MLOAD
AND       M11512	// 03.L_4th ALIGN CENTER FW
AND       P0004E	// L_4th ALIGN LEFT FW
AND       P0004D	// L_4th ALIGN CENTER FW
AND NOT   P0004C	// L_4th ALIGN SUB CENTER FW
AND NOT   P0003C	// L_4th ALIGN SUPPORT FW
AND       M04180	// R_3rd BD Z UP POS
AND       P00128	// L_4th DIE VACUUM EJECTOR ON
OUT       M11532	// STEP A¢Ò¡ÆC9
MLOAD
AND       M11513	// 04.L_4th ALIGN CENTER SUB FW
AND       P0004E	// L_4th ALIGN LEFT FW
AND       P0004D	// L_4th ALIGN CENTER FW
AND       P0004C	// L_4th ALIGN SUB CENTER FW
AND NOT   P0003C	// L_4th ALIGN SUPPORT FW
AND       M04180	// R_3rd BD Z UP POS
AND       P00128	// L_4th DIE VACUUM EJECTOR ON
OUT       M11533	// STEP A¢Ò¡ÆC10
MLOAD
AND       M11514	// 05.L_4th ROT Z 2nd
AND       P0004E	// L_4th ALIGN LEFT FW
AND       P0004D	// L_4th ALIGN CENTER FW
AND       P0004C	// L_4th ALIGN SUB CENTER FW
AND NOT   P0003C	// L_4th ALIGN SUPPORT FW
AND       M04181	// R_3rd BD Z CENTER POS
AND       P00128	// L_4th DIE VACUUM EJECTOR ON
OUT       M11534	// STEP A¢Ò¡ÆC11
MLOAD
AND       M11515	// 06.L_4th 
AND       P0004E	// L_4th ALIGN LEFT FW
AND       P0004D	// L_4th ALIGN CENTER FW
AND       P0004C	// L_4th ALIGN SUB CENTER FW
AND NOT   P0003C	// L_4th ALIGN SUPPORT FW
AND       M04181	// R_3rd BD Z CENTER POS
AND       P00128	// L_4th DIE VACUUM EJECTOR ON
OUT       M11535	// STEP A¢Ò¡ÆC12
MLOAD
AND       M11516	// 07.L_4th 
AND       P0004E	// L_4th ALIGN LEFT FW
AND       P0004D	// L_4th ALIGN CENTER FW
AND       P0004C	// L_4th ALIGN SUB CENTER FW
AND NOT   P0003C	// L_4th ALIGN SUPPORT FW
AND       M04181	// R_3rd BD Z CENTER POS
AND       P00128	// L_4th DIE VACUUM EJECTOR ON
OUT       M11536	// STEP A¢Ò¡ÆC7
MLOAD
AND       M11517	// 08.L_4th ROT Z BENDING 3rd
AND       P0004E	// L_4th ALIGN LEFT FW
AND       P0004D	// L_4th ALIGN CENTER FW
AND       P0004C	// L_4th ALIGN SUB CENTER FW
AND NOT   P0003C	// L_4th ALIGN SUPPORT FW
AND       M04182	// R_3rd BD Z BENDING POS
AND       P00128	// L_4th DIE VACUUM EJECTOR ON
OUT       M11537	// STEP A¢Ò¡ÆC8
MLOAD
AND       M11518	// 09.L_4th ROT Z BENDING 4th
AND       P0004E	// L_4th ALIGN LEFT FW
AND       P0004D	// L_4th ALIGN CENTER FW
AND       P0004C	// L_4th ALIGN SUB CENTER FW
AND NOT   P0003C	// L_4th ALIGN SUPPORT FW
AND       M04183	// 18_R_4th ROT Z BD OFFSET
AND       P00128	// L_4th DIE VACUUM EJECTOR ON
OUT       M11538	// STEP A¢Ò¡ÆC9
MLOAD
AND       M11519	// 10.L_4th SUPPORT FW
AND       P0004E	// L_4th ALIGN LEFT FW
AND       P0004D	// L_4th ALIGN CENTER FW
AND       P0004C	// L_4th ALIGN SUB CENTER FW
AND       P0003C	// L_4th ALIGN SUPPORT FW
AND       M04183	// 18_R_4th ROT Z BD OFFSET
AND       P00128	// L_4th DIE VACUUM EJECTOR ON
OUT       M11539	// STEP A¢Ò¡ÆC10
MLOAD
AND       M1151A	// 11.L_4th SUPPORT BW
AND       P0004E	// L_4th ALIGN LEFT FW
AND       P0004D	// L_4th ALIGN CENTER FW
AND       P0004C	// L_4th ALIGN SUB CENTER FW
AND NOT   P0003C	// L_4th ALIGN SUPPORT FW
AND       M04183	// 18_R_4th ROT Z BD OFFSET
AND       P00128	// L_4th DIE VACUUM EJECTOR ON
OUT       M1153A	// STEP A¢Ò¡ÆC11
MLOAD
AND       M1151B	// 12.L_4th ROT Z 1st
AND       P0004E	// L_4th ALIGN LEFT FW
AND       P0004D	// L_4th ALIGN CENTER FW
AND       P0004C	// L_4th ALIGN SUB CENTER FW
AND NOT   P0003C	// L_4th ALIGN SUPPORT FW
AND       M04180	// R_3rd BD Z UP POS
AND       P00128	// L_4th DIE VACUUM EJECTOR ON
OUT       M1153B	// STEP A¢Ò¡ÆC12
MLOAD
AND       M1151C	// 13.L_4th ALIGN CENTER SUB BW
AND       P0004E	// L_4th ALIGN LEFT FW
AND       P0004D	// L_4th ALIGN CENTER FW
AND NOT   P0004C	// L_4th ALIGN SUB CENTER FW
AND NOT   P0003C	// L_4th ALIGN SUPPORT FW
AND       M04180	// R_3rd BD Z UP POS
AND       P00128	// L_4th DIE VACUUM EJECTOR ON
OUT       M1153C	// STEP A¢Ò¡ÆC13
MLOAD
AND       M1151D	// 14.L_4th ALIGN CENTER BW/ALIGN LEFT BW
AND NOT   P0004E	// L_4th ALIGN LEFT FW
AND NOT   P0004D	// L_4th ALIGN CENTER FW
AND NOT   P0004C	// L_4th ALIGN SUB CENTER FW
AND NOT   P0003C	// L_4th ALIGN SUPPORT FW
AND       M04180	// R_3rd BD Z UP POS
AND       P00128	// L_4th DIE VACUUM EJECTOR ON
OUT       M1153D	// STEP A¢Ò¡ÆC14
MLOAD
AND       M1151E	// 15.L_4th ROT Z 1st
AND NOT   P0004E	// L_4th ALIGN LEFT FW
AND NOT   P0004D	// L_4th ALIGN CENTER FW
AND NOT   P0004C	// L_4th ALIGN SUB CENTER FW
AND NOT   P0003C	// L_4th ALIGN SUPPORT FW
AND       M04180	// R_3rd BD Z UP POS
AND       P00128	// L_4th DIE VACUUM EJECTOR ON
OUT       M1153E	// STEP A¢Ò¡ÆC15
MPOP
AND       M1151F	// 16.L_4th STEP END
OUT       M1153F	// STEP A¢Ò¡ÆC16
DMOV      32768 M1151
// output comment: 04_AU¥ì¢¯ AUAc E¢çAI

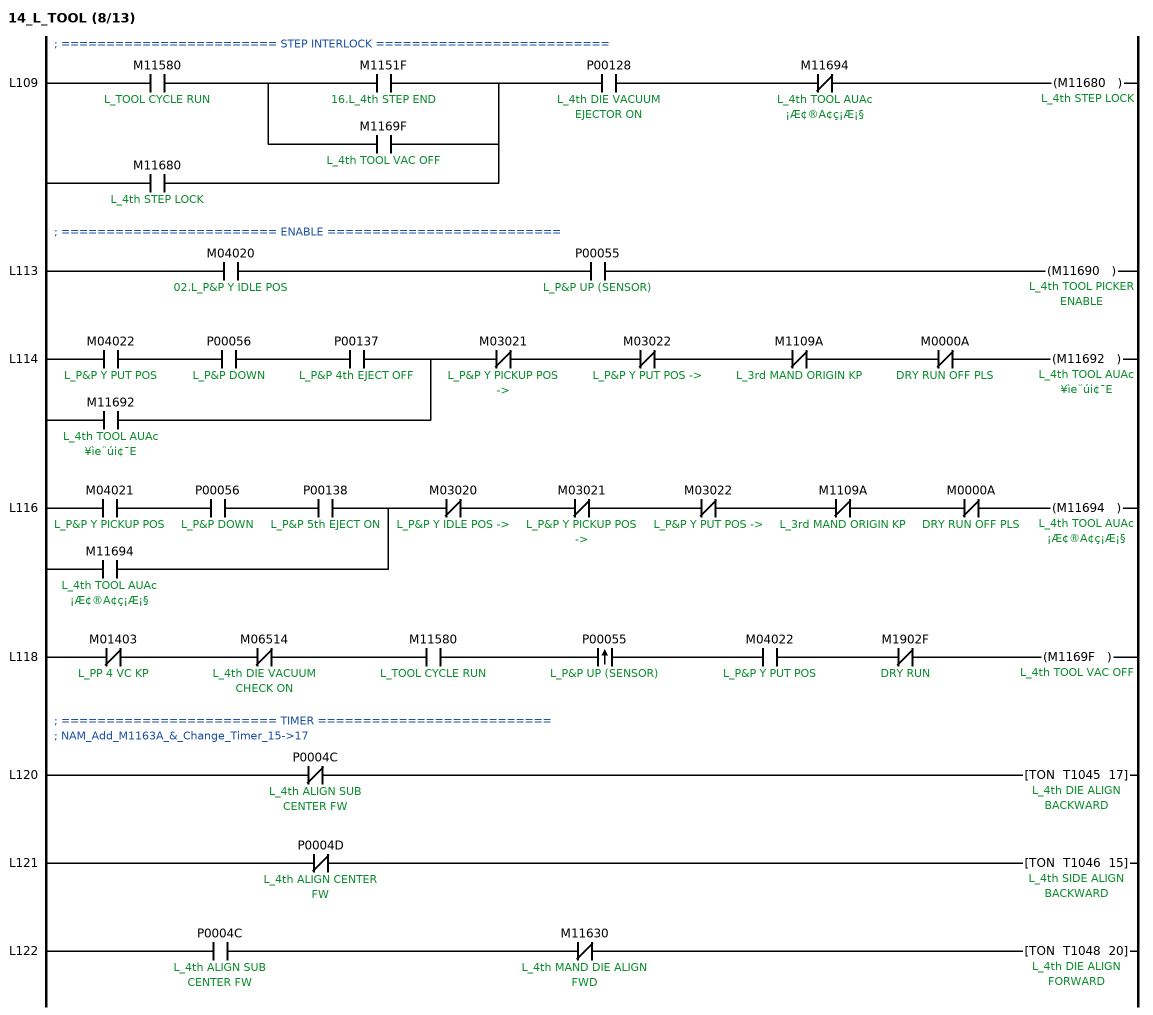
// ======================== STEP INTERLOCK ==========================
; L109
LOAD      M11580	// L_TOOL CYCLE RUN
LOAD      M1151F	// 16.L_4th STEP END
OR        M1169F	// L_4th TOOL VAC OFF
AND LOAD
OR        M11680	// L_4th STEP LOCK
AND       P00128	// L_4th DIE VACUUM EJECTOR ON
AND NOT   M11694	// L_4th TOOL AUAc ¡Æ¢®A¢ç¡Æ¡§
OUT       M11680	// L_4th STEP LOCK
// ======================== ENABLE ==========================
; L113
LOAD      M04020	// 02.L_P&P Y IDLE POS
AND       P00055	// L_P&P UP (SENSOR)
OUT       M11690	// L_4th TOOL PICKER ENABLE
; L114
LOAD      M04022	// L_P&P Y PUT POS
AND       P00056	// L_P&P DOWN
AND       P00137	// L_P&P 4th EJECT OFF
OR        M11692	// L_4th TOOL AUAc ¥ìe¨úi¢¯E
AND NOT   M03021	// L_P&P Y PICKUP POS ->
AND NOT   M03022	// L_P&P Y PUT POS ->
AND NOT   M1109A	// L_3rd MAND ORIGIN KP
AND NOT   M0000A	// DRY RUN OFF PLS
OUT       M11692	// L_4th TOOL AUAc ¥ìe¨úi¢¯E
; L116
LOAD      M04021	// L_P&P Y PICKUP POS
AND       P00056	// L_P&P DOWN
AND       P00138	// L_P&P 5th EJECT ON
OR        M11694	// L_4th TOOL AUAc ¡Æ¢®A¢ç¡Æ¡§
AND NOT   M03020	// L_P&P Y IDLE POS ->
AND NOT   M03021	// L_P&P Y PICKUP POS ->
AND NOT   M03022	// L_P&P Y PUT POS ->
AND NOT   M1109A	// L_3rd MAND ORIGIN KP
AND NOT   M0000A	// DRY RUN OFF PLS
OUT       M11694	// L_4th TOOL AUAc ¡Æ¢®A¢ç¡Æ¡§
; L118
LOAD NOT  M01403	// L_PP 4 VC KP
AND NOT   M06514	// L_4th DIE VACUUM CHECK ON
AND       M11580	// L_TOOL CYCLE RUN
ANDP      P00055	// L_P&P UP (SENSOR)
AND       M04022	// L_P&P Y PUT POS
AND NOT   M1902F	// DRY RUN
OUT       M1169F	// L_4th TOOL VAC OFF
// ======================== TIMER ==========================
; L120
LOAD NOT  P0004C	// L_4th ALIGN SUB CENTER FW
TON       T1045 17	// L_4th DIE ALIGN BACKWARD
// output comment: NAM_Add_M1163A_&_Change_Timer_15->17
; L121
LOAD NOT  P0004D	// L_4th ALIGN CENTER FW
TON       T1046 15	// L_4th SIDE ALIGN BACKWARD
; L122
LOAD      P0004C	// L_4th ALIGN SUB CENTER FW
AND NOT   M11630	// L_4th MAND DIE ALIGN FWD
TON       T1048 20	// L_4th DIE ALIGN FORWARD
// output comment: 

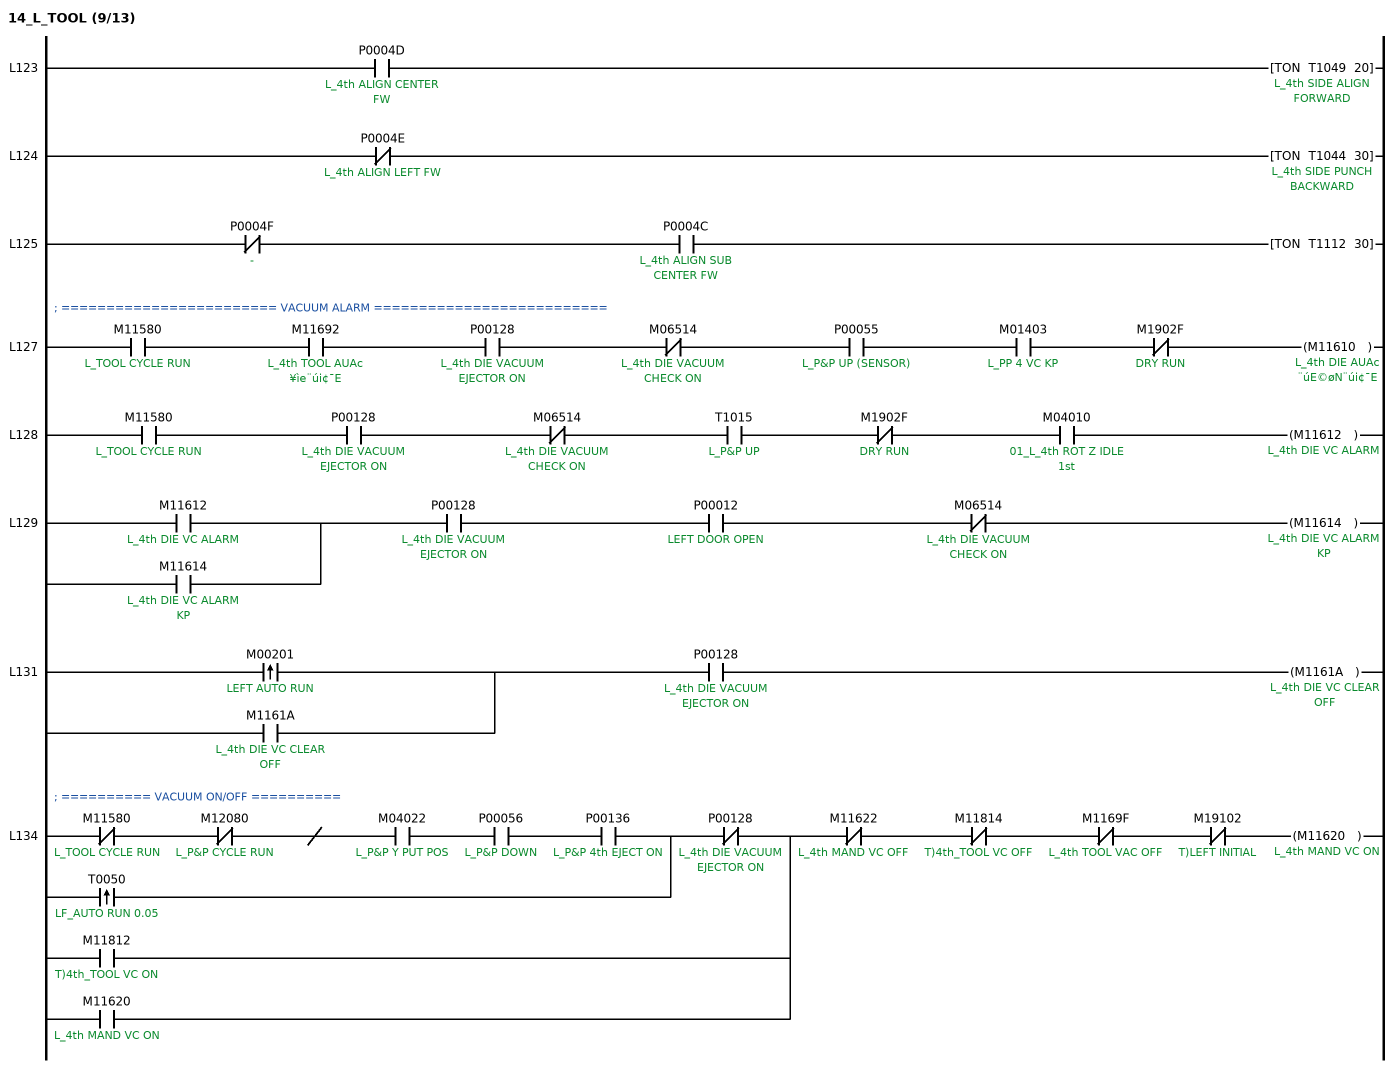
; L123
LOAD      P0004D	// L_4th ALIGN CENTER FW
TON       T1049 20	// L_4th SIDE ALIGN FORWARD
; L124
LOAD NOT  P0004E	// L_4th ALIGN LEFT FW
TON       T1044 30	// L_4th SIDE PUNCH BACKWARD
; L125
LOAD NOT  P0004F	// -
AND       P0004C	// L_4th ALIGN SUB CENTER FW
TON       T1112 30
// ======================== VACUUM ALARM ==========================
; L127
LOAD      M11580	// L_TOOL CYCLE RUN
AND       M11692	// L_4th TOOL AUAc ¥ìe¨úi¢¯E
AND       P00128	// L_4th DIE VACUUM EJECTOR ON
AND NOT   M06514	// L_4th DIE VACUUM CHECK ON
AND       P00055	// L_P&P UP (SENSOR)
AND       M01403	// L_PP 4 VC KP
AND NOT   M1902F	// DRY RUN
OUT       M11610	// L_4th DIE AUAc ¨úE©øN¨úi¢¯E
; L128
LOAD      M11580	// L_TOOL CYCLE RUN
AND       P00128	// L_4th DIE VACUUM EJECTOR ON
AND NOT   M06514	// L_4th DIE VACUUM CHECK ON
AND       T1015	// L_P&P UP
AND NOT   M1902F	// DRY RUN
AND       M04010	// 01_L_4th ROT Z IDLE 1st
OUT       M11612	// L_4th DIE VC ALARM
; L129
LOAD      M11612	// L_4th DIE VC ALARM
OR        M11614	// L_4th DIE VC ALARM KP
AND       P00128	// L_4th DIE VACUUM EJECTOR ON
AND       P00012	// LEFT DOOR OPEN
AND NOT   M06514	// L_4th DIE VACUUM CHECK ON
OUT       M11614	// L_4th DIE VC ALARM KP
; L131
LOADP     M00201	// LEFT AUTO RUN
OR        M1161A	// L_4th DIE VC CLEAR OFF
AND       P00128	// L_4th DIE VACUUM EJECTOR ON
OUT       M1161A	// L_4th DIE VC CLEAR OFF
// ========== VACUUM ON/OFF ==========
; L134
LOAD NOT  M11580	// L_TOOL CYCLE RUN
AND NOT   M12080	// L_P&P CYCLE RUN
NOT
AND       M04022	// L_P&P Y PUT POS
AND       P00056	// L_P&P DOWN
AND       P00136	// L_P&P 4th EJECT ON
ORP       T0050	// LF_AUTO RUN 0.05
AND NOT   P00128	// L_4th DIE VACUUM EJECTOR ON
OR        M11812	// T)4th_TOOL VC ON
OR        M11620	// L_4th MAND VC ON
AND NOT   M11622	// L_4th MAND VC OFF
AND NOT   M11814	// T)4th_TOOL VC OFF
AND NOT   M1169F	// L_4th TOOL VAC OFF
AND NOT   M19102	// T)LEFT INITIAL
OUT       M11620	// L_4th MAND VC ON

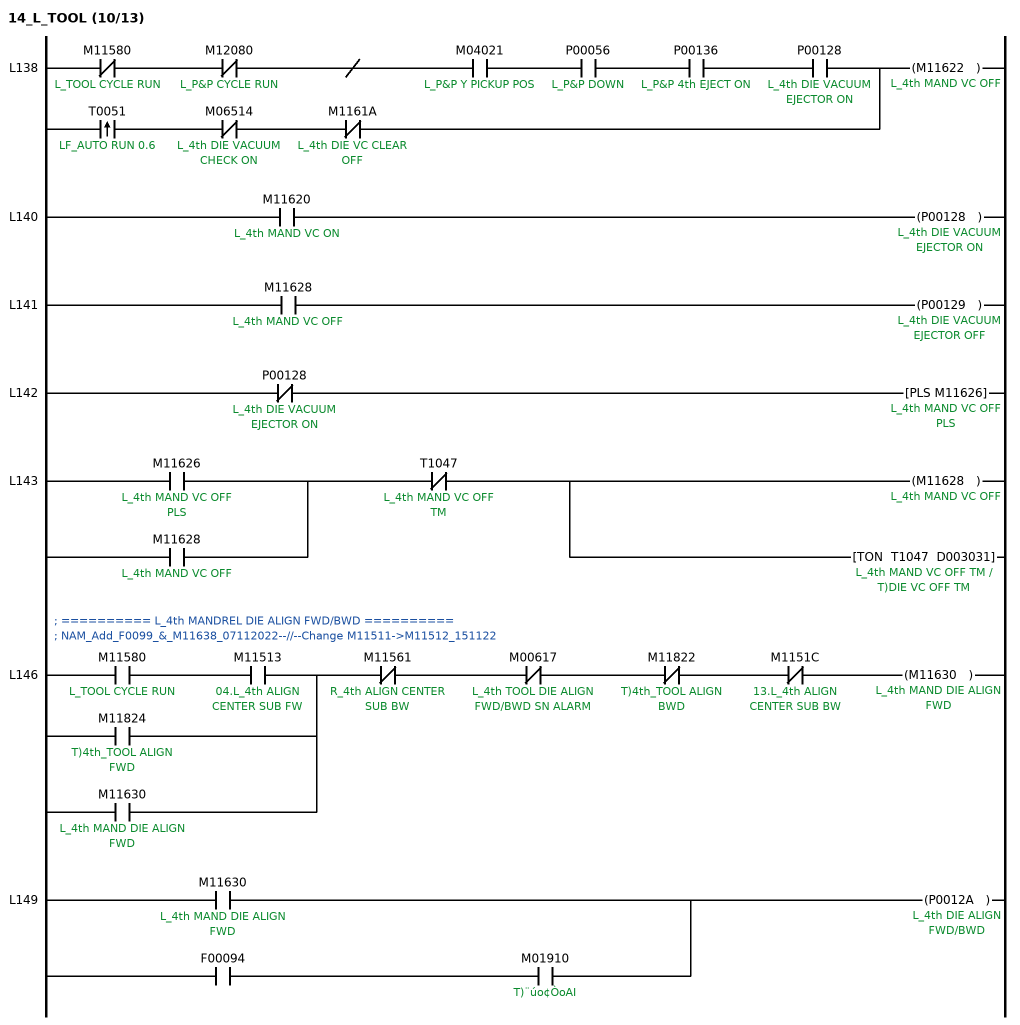
; L138
LOAD NOT  M11580	// L_TOOL CYCLE RUN
AND NOT   M12080	// L_P&P CYCLE RUN
NOT
AND       M04021	// L_P&P Y PICKUP POS
AND       P00056	// L_P&P DOWN
AND       P00136	// L_P&P 4th EJECT ON
AND       P00128	// L_4th DIE VACUUM EJECTOR ON
LOADP     T0051	// LF_AUTO RUN 0.6
AND NOT   M06514	// L_4th DIE VACUUM CHECK ON
AND NOT   M1161A	// L_4th DIE VC CLEAR OFF
OR LOAD
OUT       M11622	// L_4th MAND VC OFF
; L140
LOAD      M11620	// L_4th MAND VC ON
OUT       P00128	// L_4th DIE VACUUM EJECTOR ON
; L141
LOAD      M11628	// L_4th MAND VC OFF
OUT       P00129	// L_4th DIE VACUUM EJECTOR OFF
; L142
LOAD NOT  P00128	// L_4th DIE VACUUM EJECTOR ON
OUTP      M11626	// L_4th MAND VC OFF PLS
; L143
LOAD      M11626	// L_4th MAND VC OFF PLS
OR        M11628	// L_4th MAND VC OFF
AND NOT   T1047	// L_4th MAND VC OFF TM
OUT       M11628	// L_4th MAND VC OFF
TON       T1047 D003031	// L_4th MAND VC OFF TM / T)DIE VC OFF TM
// ========== L_4th MANDREL DIE ALIGN FWD/BWD ==========
; L146
LOAD      M11580	// L_TOOL CYCLE RUN
AND       M11513	// 04.L_4th ALIGN CENTER SUB FW
OR        M11824	// T)4th_TOOL ALIGN FWD
OR        M11630	// L_4th MAND DIE ALIGN FWD
AND NOT   M11561	// R_4th ALIGN CENTER SUB BW
AND NOT   M00617	// L_4th TOOL DIE ALIGN FWD/BWD SN ALARM
AND NOT   M11822	// T)4th_TOOL ALIGN BWD
AND NOT   M1151C	// 13.L_4th ALIGN CENTER SUB BW
OUT       M11630	// L_4th MAND DIE ALIGN FWD
// output comment: NAM_Add_F0099_&_M11638_07112022--//--Change M11511->M11512_151122
; L149
LOAD      M11630	// L_4th MAND DIE ALIGN FWD
LOAD      F00094
AND       M01910	// T)¨úo¢ÒoAI
OR LOAD
OUT       P0012A	// L_4th DIE ALIGN FWD/BWD

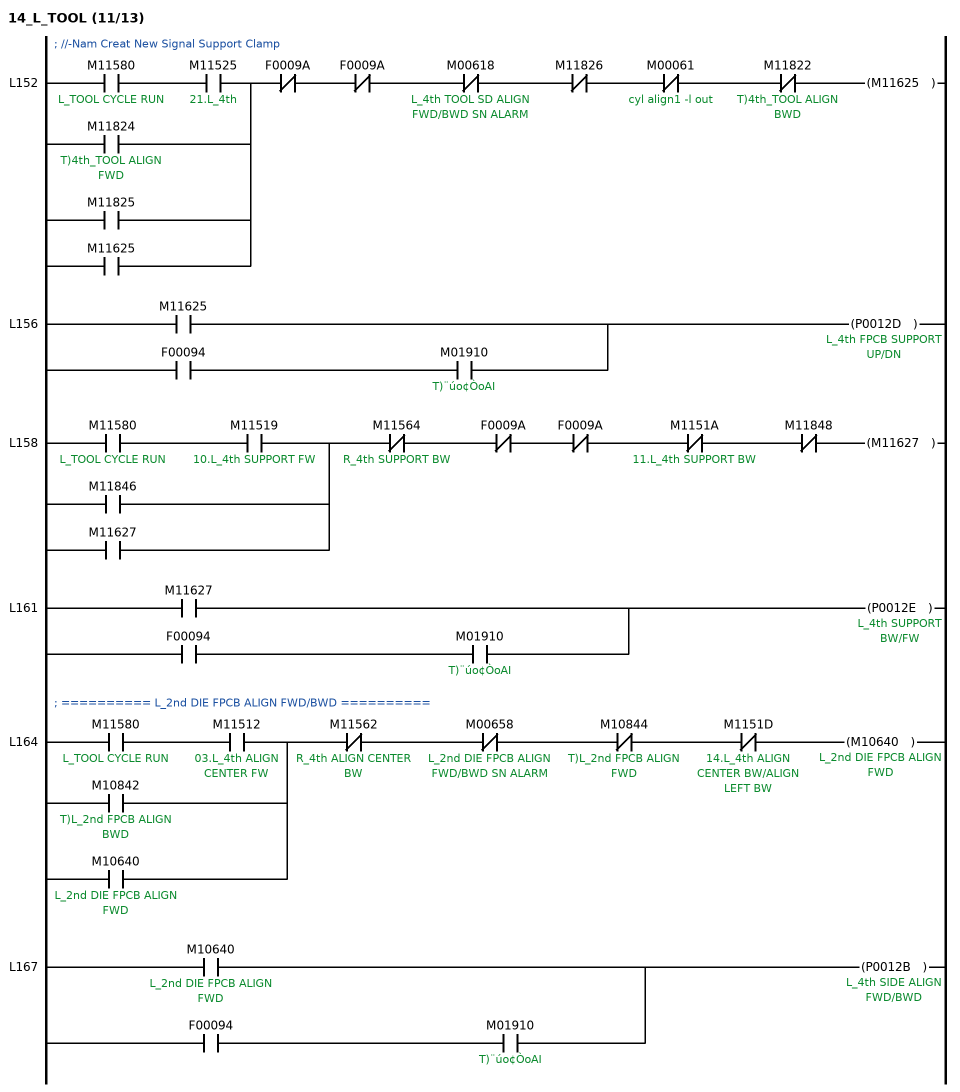
// //-Nam Creat New Signal Support Clamp
; L152
LOAD      M11580	// L_TOOL CYCLE RUN
AND       M11525	// 21.L_4th
OR        M11824	// T)4th_TOOL ALIGN FWD
OR        M11825
OR        M11625
AND NOT   F0009A
AND NOT   F0009A
AND NOT   M00618	// L_4th TOOL SD ALIGN FWD/BWD SN ALARM
AND NOT   M11826
AND NOT   M00061	// cyl align1 -l out
AND NOT   M11822	// T)4th_TOOL ALIGN BWD
OUT       M11625
; L156
LOAD      M11625
LOAD      F00094
AND       M01910	// T)¨úo¢ÒoAI
OR LOAD
OUT       P0012D	// L_4th FPCB SUPPORT UP/DN
; L158
LOAD      M11580	// L_TOOL CYCLE RUN
AND       M11519	// 10.L_4th SUPPORT FW
OR        M11846
OR        M11627
AND NOT   M11564	// R_4th SUPPORT BW
AND NOT   F0009A
AND NOT   F0009A
AND NOT   M1151A	// 11.L_4th SUPPORT BW
AND NOT   M11848
OUT       M11627
; L161
LOAD      M11627
LOAD      F00094
AND       M01910	// T)¨úo¢ÒoAI
OR LOAD
OUT       P0012E	// L_4th SUPPORT BW/FW
// ========== L_2nd DIE FPCB ALIGN FWD/BWD ==========
; L164
LOAD      M11580	// L_TOOL CYCLE RUN
AND       M11512	// 03.L_4th ALIGN CENTER FW
OR        M10842	// T)L_2nd FPCB ALIGN BWD
OR        M10640	// L_2nd DIE FPCB ALIGN FWD
AND NOT   M11562	// R_4th ALIGN CENTER BW
AND NOT   M00658	// L_2nd DIE FPCB ALIGN FWD/BWD SN ALARM
AND NOT   M10844	// T)L_2nd FPCB ALIGN FWD
AND NOT   M1151D	// 14.L_4th ALIGN CENTER BW/ALIGN LEFT BW
OUT       M10640	// L_2nd DIE FPCB ALIGN FWD
; L167
LOAD      M10640	// L_2nd DIE FPCB ALIGN FWD
LOAD      F00094
AND       M01910	// T)¨úo¢ÒoAI
OR LOAD
OUT       P0012B	// L_4th SIDE ALIGN FWD/BWD

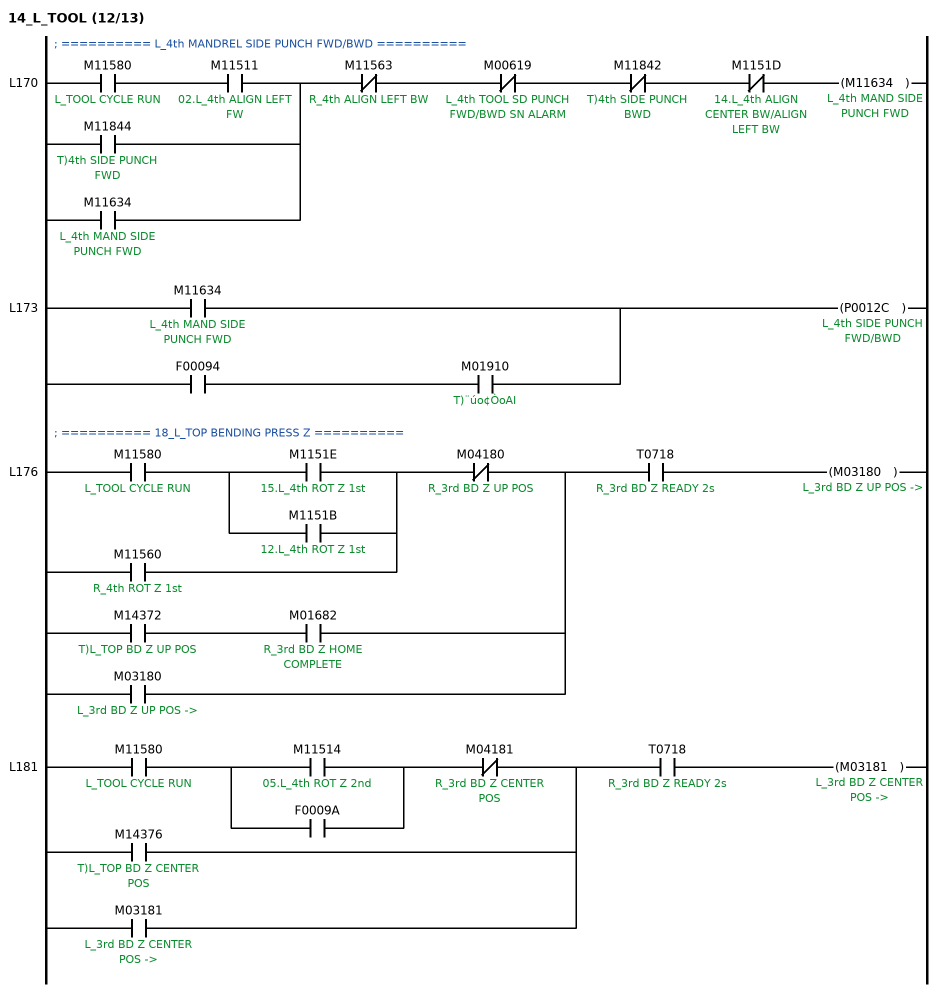
// ========== L_4th MANDREL SIDE PUNCH FWD/BWD ==========
; L170
LOAD      M11580	// L_TOOL CYCLE RUN
AND       M11511	// 02.L_4th ALIGN LEFT FW
OR        M11844	// T)4th SIDE PUNCH FWD
OR        M11634	// L_4th MAND SIDE PUNCH FWD
AND NOT   M11563	// R_4th ALIGN LEFT BW
AND NOT   M00619	// L_4th TOOL SD PUNCH FWD/BWD SN ALARM
AND NOT   M11842	// T)4th SIDE PUNCH BWD
AND NOT   M1151D	// 14.L_4th ALIGN CENTER BW/ALIGN LEFT BW
OUT       M11634	// L_4th MAND SIDE PUNCH FWD
; L173
LOAD      M11634	// L_4th MAND SIDE PUNCH FWD
LOAD      F00094
AND       M01910	// T)¨úo¢ÒoAI
OR LOAD
OUT       P0012C	// L_4th SIDE PUNCH FWD/BWD
// ========== 18_L_TOP BENDING PRESS Z ==========
; L176
LOAD      M11580	// L_TOOL CYCLE RUN
LOAD      M1151E	// 15.L_4th ROT Z 1st
OR        M1151B	// 12.L_4th ROT Z 1st
AND LOAD
OR        M11560	// R_4th ROT Z 1st
AND NOT   M04180	// R_3rd BD Z UP POS
LOAD      M14372	// T)L_TOP BD Z UP POS
AND       M01682	// R_3rd BD Z HOME COMPLETE
OR LOAD
OR        M03180	// L_3rd BD Z UP POS ->
AND       T0718	// R_3rd BD Z READY 2s
OUT       M03180	// L_3rd BD Z UP POS ->
; L181
LOAD      M11580	// L_TOOL CYCLE RUN
LOAD      M11514	// 05.L_4th ROT Z 2nd
OR        F0009A
AND LOAD
AND NOT   M04181	// R_3rd BD Z CENTER POS
OR        M14376	// T)L_TOP BD Z CENTER POS
OR        M03181	// L_3rd BD Z CENTER POS ->
AND       T0718	// R_3rd BD Z READY 2s
OUT       M03181	// L_3rd BD Z CENTER POS ->

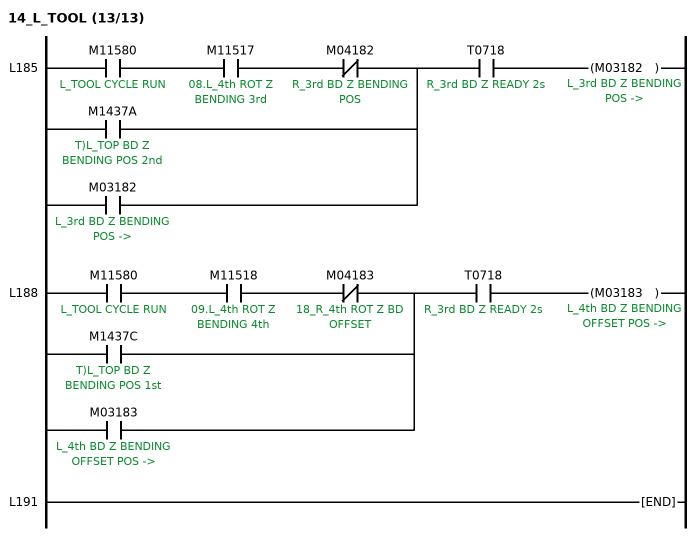
; L185
LOAD      M11580	// L_TOOL CYCLE RUN
AND       M11517	// 08.L_4th ROT Z BENDING 3rd
AND NOT   M04182	// R_3rd BD Z BENDING POS
OR        M1437A	// T)L_TOP BD Z BENDING POS 2nd
OR        M03182	// L_3rd BD Z BENDING POS ->
AND       T0718	// R_3rd BD Z READY 2s
OUT       M03182	// L_3rd BD Z BENDING POS ->
; L188
LOAD      M11580	// L_TOOL CYCLE RUN
AND       M11518	// 09.L_4th ROT Z BENDING 4th
AND NOT   M04183	// 18_R_4th ROT Z BD OFFSET
OR        M1437C	// T)L_TOP BD Z BENDING POS 1st
OR        M03183	// L_4th BD Z BENDING OFFSET POS ->
AND       T0718	// R_3rd BD Z READY 2s
OUT       M03183	// L_4th BD Z BENDING OFFSET POS ->
; L191
END

PROGRAM 15_L_PP (task: ¨ö¨¬A¥ì CA¡¤I¡¾¡¿¡¤¡Í)

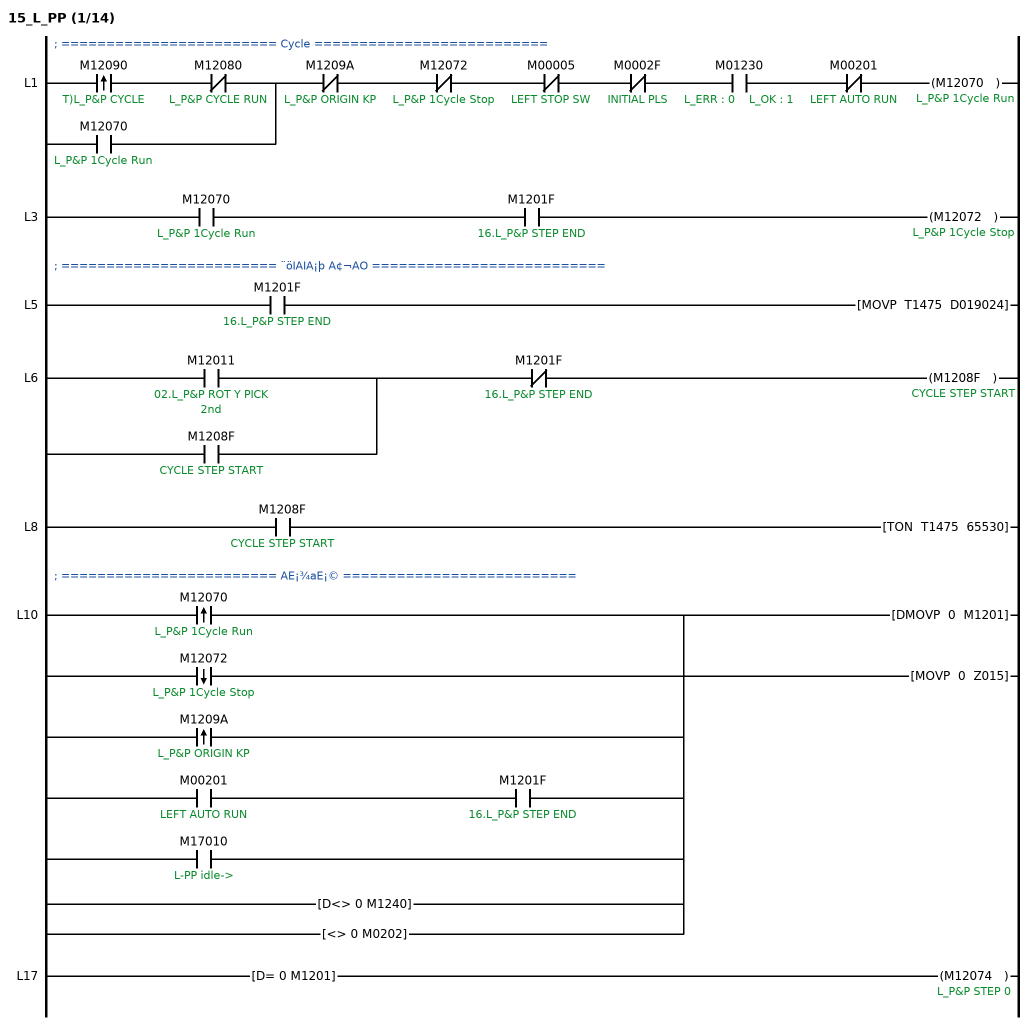
// ======================== Cycle ==========================
; L1
LOADP     M12090	// T)L_P&P CYCLE
AND NOT   M12080	// L_P&P CYCLE RUN
OR        M12070	// L_P&P 1Cycle Run
AND NOT   M1209A	// L_P&P ORIGIN KP
AND NOT   M12072	// L_P&P 1Cycle Stop
AND NOT   M00005	// LEFT STOP SW
AND NOT   M0002F	// INITIAL PLS
AND       M01230	// L_ERR : 0    L_OK : 1
AND NOT   M00201	// LEFT AUTO RUN
OUT       M12070	// L_P&P 1Cycle Run
; L3
LOAD      M12070	// L_P&P 1Cycle Run
AND       M1201F	// 16.L_P&P STEP END
OUT       M12072	// L_P&P 1Cycle Stop
// ======================== ¨öIAIA¡þ A¢¬AO ==========================
; L5
LOAD      M1201F	// 16.L_P&P STEP END
MOVP      T1475 D019024
; L6
LOAD      M12011	// 02.L_P&P ROT Y PICK 2nd
OR        M1208F	// CYCLE STEP START
AND NOT   M1201F	// 16.L_P&P STEP END
OUT       M1208F	// CYCLE STEP START
; L8
LOAD      M1208F	// CYCLE STEP START
TON       T1475 65530
// ======================== AE¡¾aE¡© ==========================
; L10
LOADP     M12070	// L_P&P 1Cycle Run
ORN       M12072	// L_P&P 1Cycle Stop
ORP       M1209A	// L_P&P ORIGIN KP
LOAD      M00201	// LEFT AUTO RUN
AND       M1201F	// 16.L_P&P STEP END
OR LOAD
OR        M17010	// L-PP idle->
ORD<>     0 M1240
OR<>      0 M0202
DMOVP     0 M1201
MOVP      0 Z015
; L17
LOADD=    0 M1201
OUT       M12074	// L_P&P STEP 0

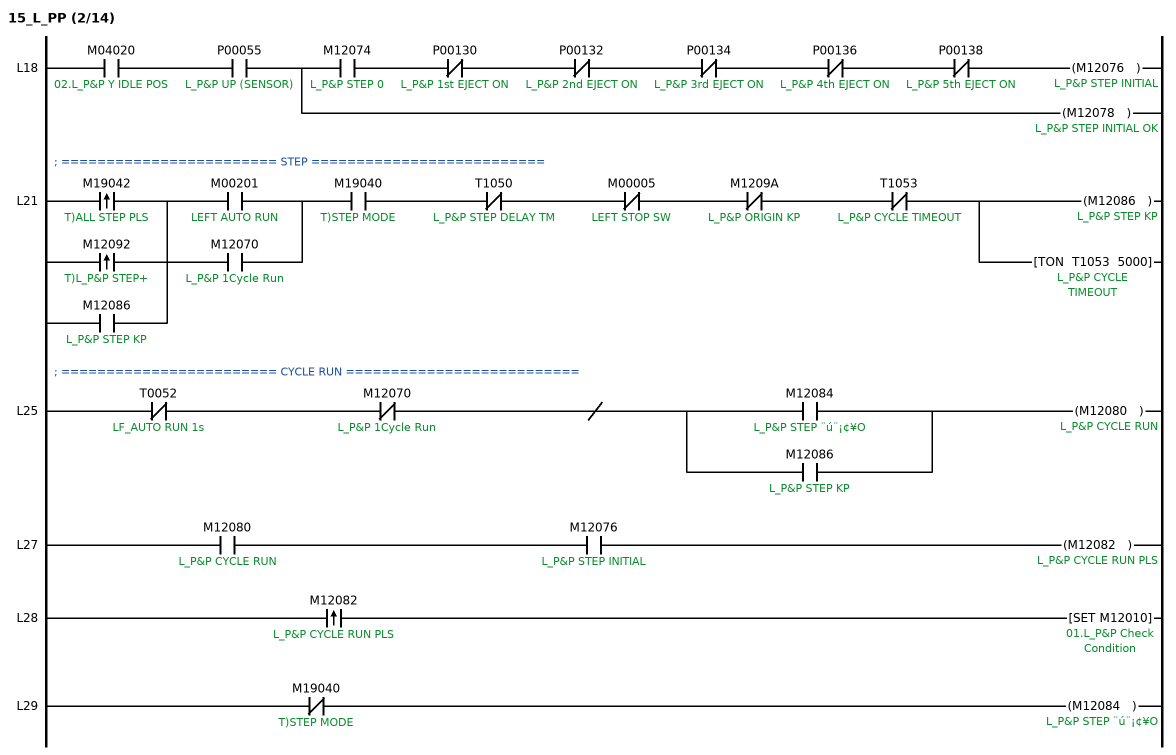
; L18
LOAD      M04020	// 02.L_P&P Y IDLE POS
AND       P00055	// L_P&P UP (SENSOR)
MPUSH
AND       M12074	// L_P&P STEP 0
AND NOT   P00130	// L_P&P 1st EJECT ON
AND NOT   P00132	// L_P&P 2nd EJECT ON
AND NOT   P00134	// L_P&P 3rd EJECT ON
AND NOT   P00136	// L_P&P 4th EJECT ON
AND NOT   P00138	// L_P&P 5th EJECT ON
OUT       M12076	// L_P&P STEP INITIAL
MPOP
OUT       M12078	// L_P&P STEP INITIAL OK
// ======================== STEP ==========================
; L21
LOADP     M19042	// T)ALL STEP PLS
ORP       M12092	// T)L_P&P STEP+
OR        M12086	// L_P&P STEP KP
LOAD      M00201	// LEFT AUTO RUN
OR        M12070	// L_P&P 1Cycle Run
AND LOAD
AND       M19040	// T)STEP MODE
AND NOT   T1050	// L_P&P STEP DELAY TM
AND NOT   M00005	// LEFT STOP SW
AND NOT   M1209A	// L_P&P ORIGIN KP
AND NOT   T1053	// L_P&P CYCLE TIMEOUT
OUT       M12086	// L_P&P STEP KP
TON       T1053 5000	// L_P&P CYCLE TIMEOUT
// ======================== CYCLE RUN ==========================
; L25
LOAD NOT  T0052	// LF_AUTO RUN 1s
AND NOT   M12070	// L_P&P 1Cycle Run
NOT
LOAD      M12084	// L_P&P STEP ¨ú¨¡¢¥O
OR        M12086	// L_P&P STEP KP
AND LOAD
OUT       M12080	// L_P&P CYCLE RUN
; L27
LOAD      M12080	// L_P&P CYCLE RUN
AND       M12076	// L_P&P STEP INITIAL
OUT       M12082	// L_P&P CYCLE RUN PLS
; L28
LOADP     M12082	// L_P&P CYCLE RUN PLS
SET       M12010	// 01.L_P&P Check Condition
; L29
LOAD NOT  M19040	// T)STEP MODE
OUT       M12084	// L_P&P STEP ¨ú¨¡¢¥O

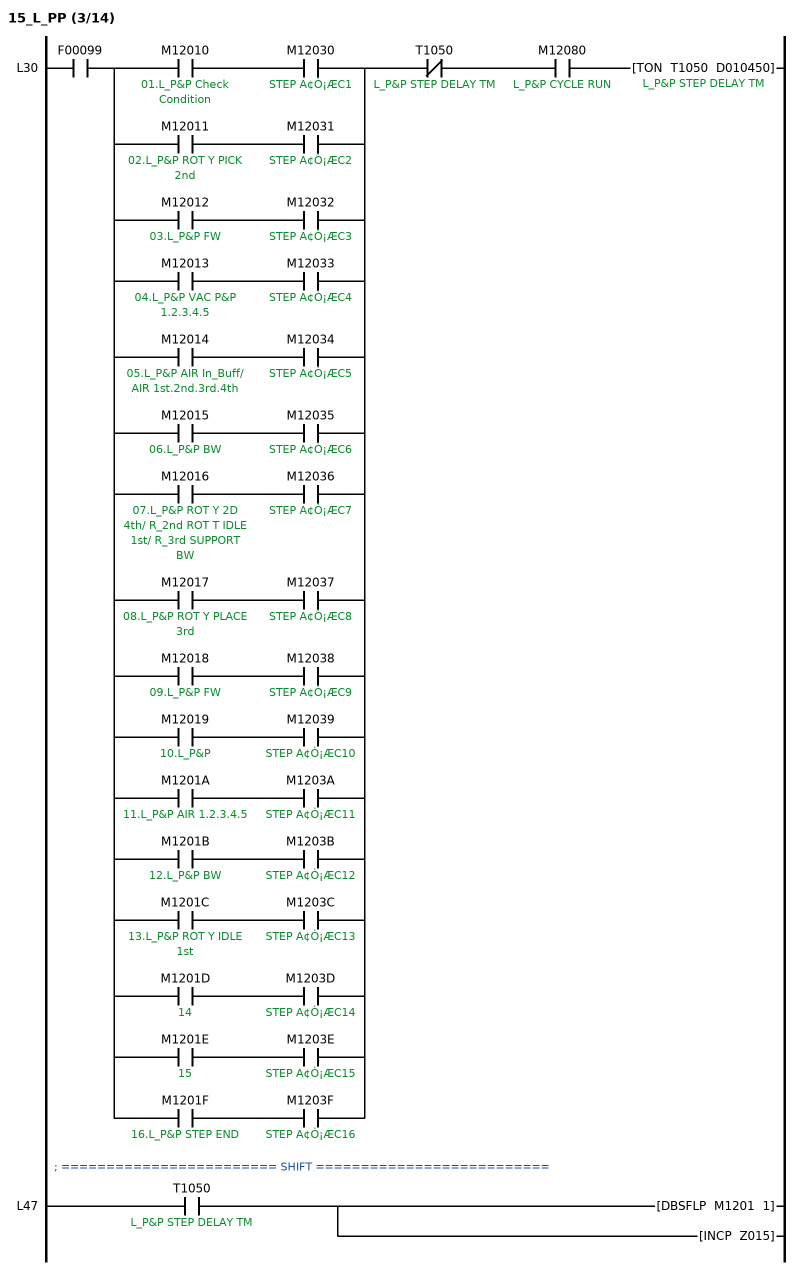
; L30
LOAD      F00099
LOAD      M12010	// 01.L_P&P Check Condition
AND       M12030	// STEP A¢Ò¡ÆC1
LOAD      M12011	// 02.L_P&P ROT Y PICK 2nd
AND       M12031	// STEP A¢Ò¡ÆC2
OR LOAD
LOAD      M12012	// 03.L_P&P FW
AND       M12032	// STEP A¢Ò¡ÆC3
OR LOAD
LOAD      M12013	// 04.L_P&P VAC P&P 1.2.3.4.5
AND       M12033	// STEP A¢Ò¡ÆC4
OR LOAD
LOAD      M12014	// 05.L_P&P AIR In_Buff/ AIR 1st.2nd.3rd.4th
AND       M12034	// STEP A¢Ò¡ÆC5
OR LOAD
LOAD      M12015	// 06.L_P&P BW
AND       M12035	// STEP A¢Ò¡ÆC6
OR LOAD
LOAD      M12016	// 07.L_P&P ROT Y 2D 4th/ R_2nd ROT T IDLE 1st/ R_3rd SUPPORT BW
AND       M12036	// STEP A¢Ò¡ÆC7
OR LOAD
LOAD      M12017	// 08.L_P&P ROT Y PLACE 3rd
AND       M12037	// STEP A¢Ò¡ÆC8
OR LOAD
LOAD      M12018	// 09.L_P&P FW
AND       M12038	// STEP A¢Ò¡ÆC9
OR LOAD
LOAD      M12019	// 10.L_P&P
AND       M12039	// STEP A¢Ò¡ÆC10
OR LOAD
LOAD      M1201A	// 11.L_P&P AIR 1.2.3.4.5
AND       M1203A	// STEP A¢Ò¡ÆC11
OR LOAD
LOAD      M1201B	// 12.L_P&P BW
AND       M1203B	// STEP A¢Ò¡ÆC12
OR LOAD
LOAD      M1201C	// 13.L_P&P ROT Y IDLE 1st
AND       M1203C	// STEP A¢Ò¡ÆC13
OR LOAD
LOAD      M1201D	// 14
AND       M1203D	// STEP A¢Ò¡ÆC14
OR LOAD
LOAD      M1201E	// 15
AND       M1203E	// STEP A¢Ò¡ÆC15
OR LOAD
LOAD      M1201F	// 16.L_P&P STEP END
AND       M1203F	// STEP A¢Ò¡ÆC16
OR LOAD
AND LOAD
AND NOT   T1050	// L_P&P STEP DELAY TM
AND       M12080	// L_P&P CYCLE RUN
TON       T1050 D010450	// L_P&P STEP DELAY TM
// ======================== SHIFT ==========================
; L47
LOAD      T1050	// L_P&P STEP DELAY TM
DBSFLP    M1201 1
INCP      Z015

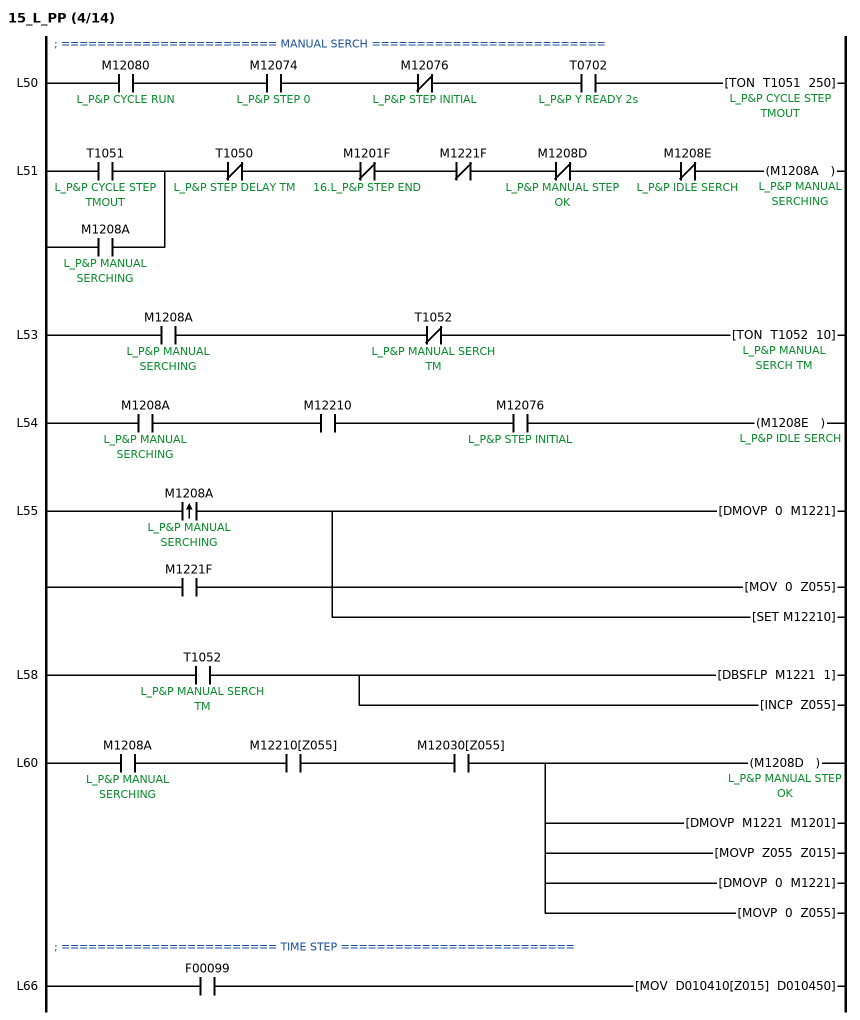
// ======================== MANUAL SERCH ==========================
; L50
LOAD      M12080	// L_P&P CYCLE RUN
AND       M12074	// L_P&P STEP 0
AND NOT   M12076	// L_P&P STEP INITIAL
AND       T0702	// L_P&P Y READY 2s
TON       T1051 250	// L_P&P CYCLE STEP TMOUT
; L51
LOAD      T1051	// L_P&P CYCLE STEP TMOUT
OR        M1208A	// L_P&P MANUAL SERCHING
AND NOT   T1050	// L_P&P STEP DELAY TM
AND NOT   M1201F	// 16.L_P&P STEP END
AND NOT   M1221F
AND NOT   M1208D	// L_P&P MANUAL STEP OK
AND NOT   M1208E	// L_P&P IDLE SERCH
OUT       M1208A	// L_P&P MANUAL SERCHING
; L53
LOAD      M1208A	// L_P&P MANUAL SERCHING
AND NOT   T1052	// L_P&P MANUAL SERCH TM
TON       T1052 10	// L_P&P MANUAL SERCH TM
; L54
LOAD      M1208A	// L_P&P MANUAL SERCHING
AND       M12210
AND       M12076	// L_P&P STEP INITIAL
OUT       M1208E	// L_P&P IDLE SERCH
; L55
LOADP     M1208A	// L_P&P MANUAL SERCHING
OR        M1221F
DMOVP     0 M1221
MOV       0 Z055
SET       M12210
; L58
LOAD      T1052	// L_P&P MANUAL SERCH TM
DBSFLP    M1221 1
INCP      Z055
; L60
LOAD      M1208A	// L_P&P MANUAL SERCHING
AND       M12210[Z055]
AND       M12030[Z055]
OUT       M1208D	// L_P&P MANUAL STEP OK
DMOVP     M1221 M1201
MOVP      Z055 Z015
DMOVP     0 M1221
MOVP      0 Z055
// ======================== TIME STEP ==========================
; L66
LOAD      F00099
MOV       D010410[Z015] D010450

